ABB RAPID module: P704.mod

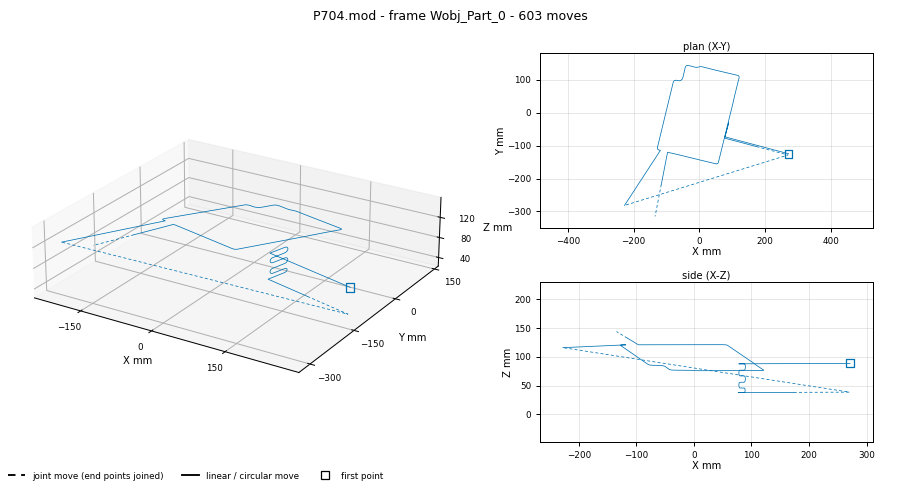
[picture p0: tool path of P704.mod in frame Wobj_Part_0, 603 of 613 moves have a stored position in this frame; points joined in program order, loops and branches not executed]
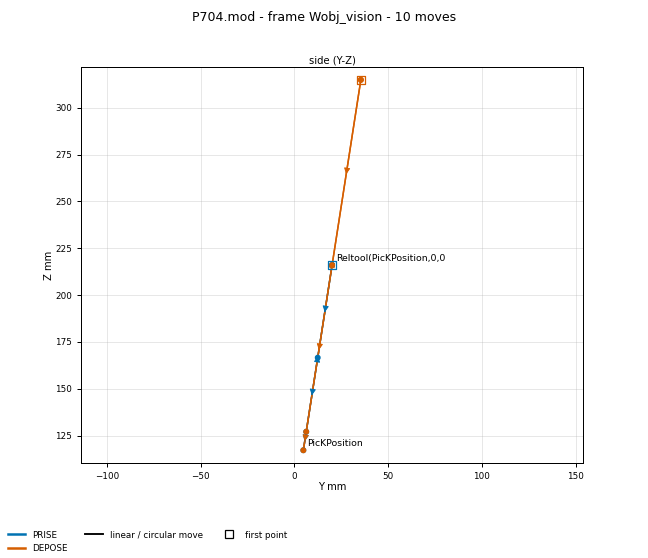
[picture p1: tool path of P704.mod in frame Wobj_vision, 10 of 613 moves have a stored position in this frame; points joined in program order, loops and branches not executed]
MODULE P704

    ! Nom         :P704
    ! Description :
    ! Créé le     :30/05/2023 09:06:17

    LOCAL CONST SPEEDDATA VitesseLente :=[10,500,0,0];
	LOCAL CONST SPEEDDATA VitesseRapide :=[30,500,0,0];
	LOCAL CONST SPEEDDATA VitesseTronconnage :=[2,500,0,0];
	LOCAL CONST SPEEDDATA VitesseTronconnageApp :=[10,500,0,0];
    !
    !Point de prise
    LOCAL PERS Robtarget PicKPosition := [[-11.2554102096367,4.78901339378507,117.207238896583],[0.0630021780734219,0.793906121478423,0.603147355662045,-0.0442387069767479],[0,0,0,0],[8.999999E+09,8.999999E+09,8.999999E+09,8.999999E+09,8.999999E+09,8.999999E+09]];
	LOCAL PERS Pose Ref := [[0,0,0],[1,0,0,0]];
    !
    !Declaration des points de meulage

    !Tr_meulage_motif_1 : Meulage d'un motif
    LOCAL CONST Robtarget Tr_meulage_motif_1_0 := [[77.98109375,-73.0847578125,87.956984375],[0.559429550316464,-0.561673578795992,-0.431884716383229,0.430159227344712],[0,0,0,0],[8.999999E+09,8.999999E+09,8.999999E+09,8.999999E+09,8.999999E+09,8.999999E+09]];
    LOCAL CONST Robtarget Tr_meulage_motif_1_1 := [[78.235953125,-72.1177734375,87.956984375],[0.559429550316464,-0.561673578795992,-0.431884716383229,0.430159227344712],[0,0,0,0],[8.999999E+09,8.999999E+09,8.999999E+09,8.999999E+09,8.999999E+09,8.999999E+09]];
    LOCAL CONST Robtarget Tr_meulage_motif_1_2 := [[78.4908046875,-71.150796875,87.956984375],[0.559429550316464,-0.561673578795992,-0.431884716383229,0.430159227344712],[0,0,0,0],[8.999999E+09,8.999999E+09,8.999999E+09,8.999999E+09,8.999999E+09,8.999999E+09]];
    LOCAL CONST Robtarget Tr_meulage_motif_1_3 := [[78.74565625,-70.1838203125,87.956984375],[0.559429550316464,-0.561673578795992,-0.431884716383229,0.430159227344712],[0,0,0,0],[8.999999E+09,8.999999E+09,8.999999E+09,8.999999E+09,8.999999E+09,8.999999E+09]];
    LOCAL CONST Robtarget Tr_meulage_motif_1_4 := [[79.0005078125,-69.2168359375,87.9569921875],[0.559429550316464,-0.561673578795992,-0.431884716383229,0.430159227344712],[0,0,0,0],[8.999999E+09,8.999999E+09,8.999999E+09,8.999999E+09,8.999999E+09,8.999999E+09]];
    LOCAL CONST Robtarget Tr_meulage_motif_1_5 := [[79.255359375,-68.249859375,87.9569921875],[0.559429550316464,-0.561673578795992,-0.431884716383229,0.430159227344712],[0,0,0,0],[8.999999E+09,8.999999E+09,8.999999E+09,8.999999E+09,8.999999E+09,8.999999E+09]];
    LOCAL CONST Robtarget Tr_meulage_motif_1_6 := [[79.51021875,-67.282875,87.9569921875],[0.559429550316464,-0.561673578795992,-0.431884716383229,0.430159227344712],[0,0,0,0],[8.999999E+09,8.999999E+09,8.999999E+09,8.999999E+09,8.999999E+09,8.999999E+09]];
    LOCAL CONST Robtarget Tr_meulage_motif_1_7 := [[79.7650703125,-66.3158984375,87.9569921875],[0.559429550316464,-0.561673578795992,-0.431884716383229,0.430159227344712],[0,0,0,0],[8.999999E+09,8.999999E+09,8.999999E+09,8.999999E+09,8.999999E+09,8.999999E+09]];
    LOCAL CONST Robtarget Tr_meulage_motif_1_8 := [[80.019921875,-65.34891796875,87.957],[0.559429550316464,-0.561673578795992,-0.431884716383229,0.430159227344712],[0,0,0,0],[8.999999E+09,8.999999E+09,8.999999E+09,8.999999E+09,8.999999E+09,8.999999E+09]];
    LOCAL CONST Robtarget Tr_meulage_motif_1_9 := [[80.2747734375,-64.38194140625,87.957],[0.559429550316464,-0.561673578795992,-0.431884716383229,0.430159227344712],[0,0,0,0],[8.999999E+09,8.999999E+09,8.999999E+09,8.999999E+09,8.999999E+09,8.999999E+09]];
    LOCAL CONST Robtarget Tr_meulage_motif_1_10 := [[80.5296328125,-63.4149609375,87.957],[0.559429550316464,-0.561673578795992,-0.431884716383229,0.430159227344712],[0,0,0,0],[8.999999E+09,8.999999E+09,8.999999E+09,8.999999E+09,8.999999E+09,8.999999E+09]];
    LOCAL CONST Robtarget Tr_meulage_motif_1_11 := [[80.784484375,-62.44798046875,87.957],[0.559429550316464,-0.561673578795992,-0.431884716383229,0.430159227344712],[0,0,0,0],[8.999999E+09,8.999999E+09,8.999999E+09,8.999999E+09,8.999999E+09,8.999999E+09]];
    LOCAL CONST Robtarget Tr_meulage_motif_1_12 := [[81.0393359375,-61.481,87.9570078125],[0.559429550316464,-0.561673578795992,-0.431884716383229,0.430159227344712],[0,0,0,0],[8.999999E+09,8.999999E+09,8.999999E+09,8.999999E+09,8.999999E+09,8.999999E+09]];
    LOCAL CONST Robtarget Tr_meulage_motif_1_13 := [[81.2941875,-60.51401953125,87.9570078125],[0.559429550316464,-0.561673578795992,-0.431884716383229,0.430159227344712],[0,0,0,0],[8.999999E+09,8.999999E+09,8.999999E+09,8.999999E+09,8.999999E+09,8.999999E+09]];
    LOCAL CONST Robtarget Tr_meulage_motif_1_14 := [[81.549046875,-59.54704296875,87.9570078125],[0.559429550316464,-0.561673578795992,-0.431884716383229,0.430159227344712],[0,0,0,0],[8.999999E+09,8.999999E+09,8.999999E+09,8.999999E+09,8.999999E+09,8.999999E+09]];
    LOCAL CONST Robtarget Tr_meulage_motif_1_15 := [[81.8038984375,-58.5800625,87.9570078125],[0.559429550316464,-0.561673578795992,-0.431884716383229,0.430159227344712],[0,0,0,0],[8.999999E+09,8.999999E+09,8.999999E+09,8.999999E+09,8.999999E+09,8.999999E+09]];
    LOCAL CONST Robtarget Tr_meulage_motif_1_16 := [[82.05875,-57.61308203125,87.957015625],[0.559429550316464,-0.561673578795992,-0.431884716383229,0.430159227344712],[0,0,0,0],[8.999999E+09,8.999999E+09,8.999999E+09,8.999999E+09,8.999999E+09,8.999999E+09]];
    LOCAL CONST Robtarget Tr_meulage_motif_1_17 := [[82.3136015625,-56.6461015625,87.957015625],[0.559429550316464,-0.561673578795992,-0.431884716383229,0.430159227344712],[0,0,0,0],[8.999999E+09,8.999999E+09,8.999999E+09,8.999999E+09,8.999999E+09,8.999999E+09]];
    LOCAL CONST Robtarget Tr_meulage_motif_1_18 := [[82.5684609375,-55.67912109375,87.957015625],[0.559429550316464,-0.561673578795992,-0.431884716383229,0.430159227344712],[0,0,0,0],[8.999999E+09,8.999999E+09,8.999999E+09,8.999999E+09,8.999999E+09,8.999999E+09]];
    LOCAL CONST Robtarget Tr_meulage_motif_1_19 := [[82.8233125,-54.712140625,87.957015625],[0.559429550316464,-0.561673578795992,-0.431884716383229,0.430159227344712],[0,0,0,0],[8.999999E+09,8.999999E+09,8.999999E+09,8.999999E+09,8.999999E+09,8.999999E+09]];
    LOCAL CONST Robtarget Tr_meulage_motif_1_20 := [[83.0781640625,-53.7451640625,87.9570234375],[0.559429550316464,-0.561673578795992,-0.431884716383229,0.430159227344712],[0,0,0,0],[8.999999E+09,8.999999E+09,8.999999E+09,8.999999E+09,8.999999E+09,8.999999E+09]];
    LOCAL CONST Robtarget Tr_meulage_motif_1_21 := [[83.333015625,-52.77818359375,87.9570234375],[0.559429550316464,-0.561673578795992,-0.431884716383229,0.430159227344712],[0,0,0,0],[8.999999E+09,8.999999E+09,8.999999E+09,8.999999E+09,8.999999E+09,8.999999E+09]];
    LOCAL CONST Robtarget Tr_meulage_motif_1_22 := [[83.587875,-51.811203125,87.9570234375],[0.559429550316464,-0.561673578795992,-0.431884716383229,0.430159227344712],[0,0,0,0],[8.999999E+09,8.999999E+09,8.999999E+09,8.999999E+09,8.999999E+09,8.999999E+09]];
    LOCAL CONST Robtarget Tr_meulage_motif_1_23 := [[83.8427265625,-50.84422265625,87.9570234375],[0.559429550316464,-0.561673578795992,-0.431884716383229,0.430159227344712],[0,0,0,0],[8.999999E+09,8.999999E+09,8.999999E+09,8.999999E+09,8.999999E+09,8.999999E+09]];
    LOCAL CONST Robtarget Tr_meulage_motif_1_24 := [[84.097578125,-49.8772421875,87.95703125],[0.559429550316464,-0.561673578795992,-0.431884716383229,0.430159227344712],[0,0,0,0],[8.999999E+09,8.999999E+09,8.999999E+09,8.999999E+09,8.999999E+09,8.999999E+09]];
    LOCAL CONST Robtarget Tr_meulage_motif_1_25 := [[84.3524296875,-48.910265625,87.95703125],[0.559429550316464,-0.561673578795992,-0.431884716383229,0.430159227344712],[0,0,0,0],[8.999999E+09,8.999999E+09,8.999999E+09,8.999999E+09,8.999999E+09,8.999999E+09]];
    LOCAL CONST Robtarget Tr_meulage_motif_1_26 := [[84.60728125,-47.94328515625,87.95703125],[0.559429550316464,-0.561673578795992,-0.431884716383229,0.430159227344712],[0,0,0,0],[8.999999E+09,8.999999E+09,8.999999E+09,8.999999E+09,8.999999E+09,8.999999E+09]];
    LOCAL CONST Robtarget Tr_meulage_motif_1_27 := [[84.862140625,-46.9763046875,87.95703125],[0.559429550316464,-0.561673578795992,-0.431884716383229,0.430159227344712],[0,0,0,0],[8.999999E+09,8.999999E+09,8.999999E+09,8.999999E+09,8.999999E+09,8.999999E+09]];
    LOCAL CONST Robtarget Tr_meulage_motif_1_28 := [[85.1169921875,-46.00932421875,87.9570390625],[0.559429550316464,-0.561673578795992,-0.431884716383229,0.430159227344712],[0,0,0,0],[8.999999E+09,8.999999E+09,8.999999E+09,8.999999E+09,8.999999E+09,8.999999E+09]];
    LOCAL CONST Robtarget Tr_meulage_motif_1_29 := [[85.37184375,-45.04234375,87.9570390625],[0.559429550316464,-0.561673578795992,-0.431884716383229,0.430159227344712],[0,0,0,0],[8.999999E+09,8.999999E+09,8.999999E+09,8.999999E+09,8.999999E+09,8.999999E+09]];
    LOCAL CONST Robtarget Tr_meulage_motif_1_30 := [[85.6266953125,-44.0753671875,87.9570390625],[0.559429550316464,-0.561673578795992,-0.431884716383229,0.430159227344712],[0,0,0,0],[8.999999E+09,8.999999E+09,8.999999E+09,8.999999E+09,8.999999E+09,8.999999E+09]];
    LOCAL CONST Robtarget Tr_meulage_motif_1_31 := [[85.8815546875,-43.10838671875,87.9570390625],[0.559429550316464,-0.561673578795992,-0.431884716383229,0.430159227344712],[0,0,0,0],[8.999999E+09,8.999999E+09,8.999999E+09,8.999999E+09,8.999999E+09,8.999999E+09]];
    LOCAL CONST Robtarget Tr_meulage_motif_1_32 := [[86.13640625,-42.14140625,87.957046875],[0.559429550316464,-0.561673578795992,-0.431884716383229,0.430159227344712],[0,0,0,0],[8.999999E+09,8.999999E+09,8.999999E+09,8.999999E+09,8.999999E+09,8.999999E+09]];
    LOCAL CONST Robtarget Tr_meulage_motif_1_33 := [[86.3912578125,-41.17442578125,87.957046875],[0.559429550316464,-0.561673578795992,-0.431884716383229,0.430159227344712],[0,0,0,0],[8.999999E+09,8.999999E+09,8.999999E+09,8.999999E+09,8.999999E+09,8.999999E+09]];
    LOCAL CONST Robtarget Tr_meulage_motif_1_34 := [[86.646109375,-40.2074453125,87.957046875],[0.559429550316464,-0.561673578795992,-0.431884716383229,0.430159227344712],[0,0,0,0],[8.999999E+09,8.999999E+09,8.999999E+09,8.999999E+09,8.999999E+09,8.999999E+09]];
    LOCAL CONST Robtarget Tr_meulage_motif_1_35 := [[86.90096875,-39.24046875,87.957046875],[0.559429550316464,-0.561673578795992,-0.431884716383229,0.430159227344712],[0,0,0,0],[8.999999E+09,8.999999E+09,8.999999E+09,8.999999E+09,8.999999E+09,8.999999E+09]];
    LOCAL CONST Robtarget Tr_meulage_motif_1_36 := [[87.1558203125,-38.27348828125,87.9570546875],[0.559429550316464,-0.561673578795992,-0.431884716383229,0.430159227344712],[0,0,0,0],[8.999999E+09,8.999999E+09,8.999999E+09,8.999999E+09,8.999999E+09,8.999999E+09]];
    LOCAL CONST Robtarget Tr_meulage_motif_1_37 := [[87.410671875,-37.3065078125,87.9570546875],[0.559429550316464,-0.561673578795992,-0.431884716383229,0.430159227344712],[0,0,0,0],[8.999999E+09,8.999999E+09,8.999999E+09,8.999999E+09,8.999999E+09,8.999999E+09]];
    LOCAL CONST Robtarget Tr_meulage_motif_1_38 := [[87.6655234375,-36.33952734375,87.9570546875],[0.559429550316464,-0.561673578795992,-0.431884716383229,0.430159227344712],[0,0,0,0],[8.999999E+09,8.999999E+09,8.999999E+09,8.999999E+09,8.999999E+09,8.999999E+09]];
    LOCAL CONST Robtarget Tr_meulage_motif_1_39 := [[87.9182109375,-35.37966796875,87.8464609375],[0.559429550316464,-0.561673578795992,-0.431884716383229,0.430159227344712],[0,0,0,0],[8.999999E+09,8.999999E+09,8.999999E+09,8.999999E+09,8.999999E+09,8.999999E+09]];
    LOCAL CONST Robtarget Tr_meulage_motif_1_40 := [[88.158921875,-34.4642890625,87.63528125],[0.559429550316464,-0.561673578795992,-0.431884716383229,0.430159227344712],[0,0,0,0],[8.999999E+09,8.999999E+09,8.999999E+09,8.999999E+09,8.999999E+09,8.999999E+09]];
    LOCAL CONST Robtarget Tr_meulage_motif_1_41 := [[88.375578125,-33.63955078125,87.3634375],[0.559429550316464,-0.561673578795992,-0.431884716383229,0.430159227344712],[0,0,0,0],[8.999999E+09,8.999999E+09,8.999999E+09,8.999999E+09,8.999999E+09,8.999999E+09]];
    LOCAL CONST Robtarget Tr_meulage_motif_1_42 := [[88.56603125,-32.91419921875,87.0875],[0.559429550316464,-0.561673578795992,-0.431884716383229,0.430159227344712],[0,0,0,0],[8.999999E+09,8.999999E+09,8.999999E+09,8.999999E+09,8.999999E+09,8.999999E+09]];
    LOCAL CONST Robtarget Tr_meulage_motif_1_43 := [[88.845140625,-31.84909765625,86.4713828125],[0.559429550316464,-0.561673578795992,-0.431884716383229,0.430159227344712],[0,0,0,0],[8.999999E+09,8.999999E+09,8.999999E+09,8.999999E+09,8.999999E+09,8.999999E+09]];
    LOCAL CONST Robtarget Tr_meulage_motif_1_44 := [[89.104015625,-30.858484375,85.623734375],[0.559429550316464,-0.561673578795992,-0.431884716383229,0.430159227344712],[0,0,0,0],[8.999999E+09,8.999999E+09,8.999999E+09,8.999999E+09,8.999999E+09,8.999999E+09]];
    LOCAL CONST Robtarget Tr_meulage_motif_1_45 := [[89.317546875,-30.03816015625,84.599859375],[0.559429550316464,-0.561673578795992,-0.431884716383229,0.430159227344712],[0,0,0,0],[8.999999E+09,8.999999E+09,8.999999E+09,8.999999E+09,8.999999E+09,8.999999E+09]];
    LOCAL CONST Robtarget Tr_meulage_motif_1_46 := [[89.4392421875,-29.565404296875,83.4836796875],[0.559429550316464,-0.561673578795992,-0.431884716383229,0.430159227344712],[0,0,0,0],[8.999999E+09,8.999999E+09,8.999999E+09,8.999999E+09,8.999999E+09,8.999999E+09]];
    LOCAL CONST Robtarget Tr_meulage_motif_1_47 := [[89.4444453125,-29.538787109375,82.7877109375],[0.559429550316464,-0.561673578795992,-0.431884716383229,0.430159227344712],[0,0,0,0],[8.999999E+09,8.999999E+09,8.999999E+09,8.999999E+09,8.999999E+09,8.999999E+09]];
    LOCAL CONST Robtarget Tr_meulage_motif_1_48 := [[89.4428359375,-29.538361328125,82.1264609375],[0.559429550316464,-0.561673578795992,-0.431884716383229,0.430159227344712],[0,0,0,0],[8.999999E+09,8.999999E+09,8.999999E+09,8.999999E+09,8.999999E+09,8.999999E+09]];
    LOCAL CONST Robtarget Tr_meulage_motif_1_49 := [[89.427234375,-29.591,81.465375],[0.559429550316464,-0.561673578795992,-0.431884716383229,0.430159227344712],[0,0,0,0],[8.999999E+09,8.999999E+09,8.999999E+09,8.999999E+09,8.999999E+09,8.999999E+09]];
    LOCAL CONST Robtarget Tr_meulage_motif_1_50 := [[89.2975859375,-30.07205859375,80.363625],[0.559429550316464,-0.561673578795992,-0.431884716383229,0.430159227344712],[0,0,0,0],[8.999999E+09,8.999999E+09,8.999999E+09,8.999999E+09,8.999999E+09,8.999999E+09]];
    LOCAL CONST Robtarget Tr_meulage_motif_1_51 := [[89.0768203125,-30.899748046875,79.357],[0.559429550316464,-0.561673578795992,-0.431884716383229,0.430159227344712],[0,0,0,0],[8.999999E+09,8.999999E+09,8.999999E+09,8.999999E+09,8.999999E+09,8.999999E+09]];
    LOCAL CONST Robtarget Tr_meulage_motif_1_52 := [[88.813984375,-31.888828125,78.528125],[0.559429550316464,-0.561673578795992,-0.431884716383229,0.430159227344712],[0,0,0,0],[8.999999E+09,8.999999E+09,8.999999E+09,8.999999E+09,8.999999E+09,8.999999E+09]];
    LOCAL CONST Robtarget Tr_meulage_motif_1_53 := [[88.6379140625,-32.552978515625,78.132375],[0.559429550316464,-0.561673578795992,-0.431884716383229,0.430159227344712],[0,0,0,0],[8.999999E+09,8.999999E+09,8.999999E+09,8.999999E+09,8.999999E+09,8.999999E+09]];
    LOCAL CONST Robtarget Tr_meulage_motif_1_54 := [[88.3415625,-33.672578125,77.64484375],[0.559429550316464,-0.561673578795992,-0.431884716383229,0.430159227344712],[0,0,0,0],[8.999999E+09,8.999999E+09,8.999999E+09,8.999999E+09,8.999999E+09,8.999999E+09]];
    LOCAL CONST Robtarget Tr_meulage_motif_1_55 := [[88.1255625,-34.4895390625,77.38075],[0.559429550316464,-0.561673578795992,-0.431884716383229,0.430159227344712],[0,0,0,0],[8.999999E+09,8.999999E+09,8.999999E+09,8.999999E+09,8.999999E+09,8.999999E+09]];
    LOCAL CONST Robtarget Tr_meulage_motif_1_56 := [[87.8875390625,-35.39062890625,77.17628125],[0.559429550316464,-0.561673578795992,-0.431884716383229,0.430159227344712],[0,0,0,0],[8.999999E+09,8.999999E+09,8.999999E+09,8.999999E+09,8.999999E+09,8.999999E+09]];
    LOCAL CONST Robtarget Tr_meulage_motif_1_57 := [[87.637125,-36.3397109375,77.0676875],[0.559429550316464,-0.561673578795992,-0.431884716383229,0.430159227344712],[0,0,0,0],[8.999999E+09,8.999999E+09,8.999999E+09,8.999999E+09,8.999999E+09,8.999999E+09]];
    LOCAL CONST Robtarget Tr_meulage_motif_1_58 := [[87.3838984375,-37.2994296875,76.9570859375],[0.559429550316464,-0.561673578795992,-0.431884716383229,0.430159227344712],[0,0,0,0],[8.999999E+09,8.999999E+09,8.999999E+09,8.999999E+09,8.999999E+09,8.999999E+09]];
    LOCAL CONST Robtarget Tr_meulage_motif_1_59 := [[87.1290390625,-38.26641015625,76.9570859375],[0.559429550316464,-0.561673578795992,-0.431884716383229,0.430159227344712],[0,0,0,0],[8.999999E+09,8.999999E+09,8.999999E+09,8.999999E+09,8.999999E+09,8.999999E+09]];
    LOCAL CONST Robtarget Tr_meulage_motif_1_60 := [[86.8741875,-39.23338671875,76.9570859375],[0.559429550316464,-0.561673578795992,-0.431884716383229,0.430159227344712],[0,0,0,0],[8.999999E+09,8.999999E+09,8.999999E+09,8.999999E+09,8.999999E+09,8.999999E+09]];
    LOCAL CONST Robtarget Tr_meulage_motif_1_61 := [[86.6193359375,-40.2003671875,76.9570859375],[0.559429550316464,-0.561673578795992,-0.431884716383229,0.430159227344712],[0,0,0,0],[8.999999E+09,8.999999E+09,8.999999E+09,8.999999E+09,8.999999E+09,8.999999E+09]];
    LOCAL CONST Robtarget Tr_meulage_motif_1_62 := [[86.364484375,-41.16734765625,76.957078125],[0.559429550316464,-0.561673578795992,-0.431884716383229,0.430159227344712],[0,0,0,0],[8.999999E+09,8.999999E+09,8.999999E+09,8.999999E+09,8.999999E+09,8.999999E+09]];
    LOCAL CONST Robtarget Tr_meulage_motif_1_63 := [[86.109625,-42.134328125,76.957078125],[0.559429550316464,-0.561673578795992,-0.431884716383229,0.430159227344712],[0,0,0,0],[8.999999E+09,8.999999E+09,8.999999E+09,8.999999E+09,8.999999E+09,8.999999E+09]];
    LOCAL CONST Robtarget Tr_meulage_motif_1_64 := [[85.8547734375,-43.10130859375,76.957078125],[0.559429550316464,-0.561673578795992,-0.431884716383229,0.430159227344712],[0,0,0,0],[8.999999E+09,8.999999E+09,8.999999E+09,8.999999E+09,8.999999E+09,8.999999E+09]];
    LOCAL CONST Robtarget Tr_meulage_motif_1_65 := [[85.599921875,-44.06828515625,76.957078125],[0.559429550316464,-0.561673578795992,-0.431884716383229,0.430159227344712],[0,0,0,0],[8.999999E+09,8.999999E+09,8.999999E+09,8.999999E+09,8.999999E+09,8.999999E+09]];
    LOCAL CONST Robtarget Tr_meulage_motif_1_66 := [[85.3450703125,-45.035265625,76.9570703125],[0.559429550316464,-0.561673578795992,-0.431884716383229,0.430159227344712],[0,0,0,0],[8.999999E+09,8.999999E+09,8.999999E+09,8.999999E+09,8.999999E+09,8.999999E+09]];
    LOCAL CONST Robtarget Tr_meulage_motif_1_67 := [[85.0902109375,-46.00224609375,76.9570703125],[0.559429550316464,-0.561673578795992,-0.431884716383229,0.430159227344712],[0,0,0,0],[8.999999E+09,8.999999E+09,8.999999E+09,8.999999E+09,8.999999E+09,8.999999E+09]];
    LOCAL CONST Robtarget Tr_meulage_motif_1_68 := [[84.835359375,-46.9692265625,76.9570703125],[0.559429550316464,-0.561673578795992,-0.431884716383229,0.430159227344712],[0,0,0,0],[8.999999E+09,8.999999E+09,8.999999E+09,8.999999E+09,8.999999E+09,8.999999E+09]];
    LOCAL CONST Robtarget Tr_meulage_motif_1_69 := [[84.5805078125,-47.93620703125,76.9570703125],[0.559429550316464,-0.561673578795992,-0.431884716383229,0.430159227344712],[0,0,0,0],[8.999999E+09,8.999999E+09,8.999999E+09,8.999999E+09,8.999999E+09,8.999999E+09]];
    LOCAL CONST Robtarget Tr_meulage_motif_1_70 := [[84.32565625,-48.90318359375,76.9570625],[0.559429550316464,-0.561673578795992,-0.431884716383229,0.430159227344712],[0,0,0,0],[8.999999E+09,8.999999E+09,8.999999E+09,8.999999E+09,8.999999E+09,8.999999E+09]];
    LOCAL CONST Robtarget Tr_meulage_motif_1_71 := [[84.070796875,-49.8701640625,76.9570625],[0.559429550316464,-0.561673578795992,-0.431884716383229,0.430159227344712],[0,0,0,0],[8.999999E+09,8.999999E+09,8.999999E+09,8.999999E+09,8.999999E+09,8.999999E+09]];
    LOCAL CONST Robtarget Tr_meulage_motif_1_72 := [[83.8159453125,-50.83714453125,76.9570625],[0.559429550316464,-0.561673578795992,-0.431884716383229,0.430159227344712],[0,0,0,0],[8.999999E+09,8.999999E+09,8.999999E+09,8.999999E+09,8.999999E+09,8.999999E+09]];
    LOCAL CONST Robtarget Tr_meulage_motif_1_73 := [[83.56109375,-51.804125,76.9570625],[0.559429550316464,-0.561673578795992,-0.431884716383229,0.430159227344712],[0,0,0,0],[8.999999E+09,8.999999E+09,8.999999E+09,8.999999E+09,8.999999E+09,8.999999E+09]];
    LOCAL CONST Robtarget Tr_meulage_motif_1_74 := [[83.3062421875,-52.77110546875,76.9570546875],[0.559429550316464,-0.561673578795992,-0.431884716383229,0.430159227344712],[0,0,0,0],[8.999999E+09,8.999999E+09,8.999999E+09,8.999999E+09,8.999999E+09,8.999999E+09]];
    LOCAL CONST Robtarget Tr_meulage_motif_1_75 := [[83.051390625,-53.73808203125,76.9570546875],[0.559429550316464,-0.561673578795992,-0.431884716383229,0.430159227344712],[0,0,0,0],[8.999999E+09,8.999999E+09,8.999999E+09,8.999999E+09,8.999999E+09,8.999999E+09]];
    LOCAL CONST Robtarget Tr_meulage_motif_1_76 := [[82.79653125,-54.7050625,76.9570546875],[0.559429550316464,-0.561673578795992,-0.431884716383229,0.430159227344712],[0,0,0,0],[8.999999E+09,8.999999E+09,8.999999E+09,8.999999E+09,8.999999E+09,8.999999E+09]];
    LOCAL CONST Robtarget Tr_meulage_motif_1_77 := [[82.5416796875,-55.67204296875,76.9570546875],[0.559429550316464,-0.561673578795992,-0.431884716383229,0.430159227344712],[0,0,0,0],[8.999999E+09,8.999999E+09,8.999999E+09,8.999999E+09,8.999999E+09,8.999999E+09]];
    LOCAL CONST Robtarget Tr_meulage_motif_1_78 := [[82.286828125,-56.6390234375,76.957046875],[0.559429550316464,-0.561673578795992,-0.431884716383229,0.430159227344712],[0,0,0,0],[8.999999E+09,8.999999E+09,8.999999E+09,8.999999E+09,8.999999E+09,8.999999E+09]];
    LOCAL CONST Robtarget Tr_meulage_motif_1_79 := [[82.0319765625,-57.60600390625,76.957046875],[0.559429550316464,-0.561673578795992,-0.431884716383229,0.430159227344712],[0,0,0,0],[8.999999E+09,8.999999E+09,8.999999E+09,8.999999E+09,8.999999E+09,8.999999E+09]];
    LOCAL CONST Robtarget Tr_meulage_motif_1_80 := [[81.7771171875,-58.57298046875,76.957046875],[0.559429550316464,-0.561673578795992,-0.431884716383229,0.430159227344712],[0,0,0,0],[8.999999E+09,8.999999E+09,8.999999E+09,8.999999E+09,8.999999E+09,8.999999E+09]];
    LOCAL CONST Robtarget Tr_meulage_motif_1_81 := [[81.522265625,-59.5399609375,76.957046875],[0.559429550316464,-0.561673578795992,-0.431884716383229,0.430159227344712],[0,0,0,0],[8.999999E+09,8.999999E+09,8.999999E+09,8.999999E+09,8.999999E+09,8.999999E+09]];
    LOCAL CONST Robtarget Tr_meulage_motif_1_82 := [[81.2674140625,-60.50694140625,76.9570390625],[0.559429550316464,-0.561673578795992,-0.431884716383229,0.430159227344712],[0,0,0,0],[8.999999E+09,8.999999E+09,8.999999E+09,8.999999E+09,8.999999E+09,8.999999E+09]];
    LOCAL CONST Robtarget Tr_meulage_motif_1_83 := [[81.0125625,-61.473921875,76.9570390625],[0.559429550316464,-0.561673578795992,-0.431884716383229,0.430159227344712],[0,0,0,0],[8.999999E+09,8.999999E+09,8.999999E+09,8.999999E+09,8.999999E+09,8.999999E+09]];
    LOCAL CONST Robtarget Tr_meulage_motif_1_84 := [[80.757703125,-62.44090234375,76.9570390625],[0.559429550316464,-0.561673578795992,-0.431884716383229,0.430159227344712],[0,0,0,0],[8.999999E+09,8.999999E+09,8.999999E+09,8.999999E+09,8.999999E+09,8.999999E+09]];
    LOCAL CONST Robtarget Tr_meulage_motif_1_85 := [[80.5028515625,-63.40787890625,76.9570390625],[0.559429550316464,-0.561673578795992,-0.431884716383229,0.430159227344712],[0,0,0,0],[8.999999E+09,8.999999E+09,8.999999E+09,8.999999E+09,8.999999E+09,8.999999E+09]];
    LOCAL CONST Robtarget Tr_meulage_motif_1_86 := [[80.248,-64.374859375,76.95703125],[0.559429550316464,-0.561673578795992,-0.431884716383229,0.430159227344712],[0,0,0,0],[8.999999E+09,8.999999E+09,8.999999E+09,8.999999E+09,8.999999E+09,8.999999E+09]];
    LOCAL CONST Robtarget Tr_meulage_motif_1_87 := [[79.9931484375,-65.34183984375,76.95703125],[0.559429550316464,-0.561673578795992,-0.431884716383229,0.430159227344712],[0,0,0,0],[8.999999E+09,8.999999E+09,8.999999E+09,8.999999E+09,8.999999E+09,8.999999E+09]];
    LOCAL CONST Robtarget Tr_meulage_motif_1_88 := [[79.7382890625,-66.3088203125,76.95703125],[0.559429550316464,-0.561673578795992,-0.431884716383229,0.430159227344712],[0,0,0,0],[8.999999E+09,8.999999E+09,8.999999E+09,8.999999E+09,8.999999E+09,8.999999E+09]];
    LOCAL CONST Robtarget Tr_meulage_motif_1_89 := [[79.4850625,-67.2685390625,76.8464375],[0.559429550316464,-0.561673578795992,-0.431884716383229,0.430159227344712],[0,0,0,0],[8.999999E+09,8.999999E+09,8.999999E+09,8.999999E+09,8.999999E+09,8.999999E+09]];
    LOCAL CONST Robtarget Tr_meulage_motif_1_90 := [[79.2433359375,-68.1836484375,76.63525],[0.559429550316464,-0.561673578795992,-0.431884716383229,0.430159227344712],[0,0,0,0],[8.999999E+09,8.999999E+09,8.999999E+09,8.999999E+09,8.999999E+09,8.999999E+09]];
    LOCAL CONST Robtarget Tr_meulage_motif_1_91 := [[79.0253515625,-69.00803125,76.36340625],[0.559429550316464,-0.561673578795992,-0.431884716383229,0.430159227344712],[0,0,0,0],[8.999999E+09,8.999999E+09,8.999999E+09,8.999999E+09,8.999999E+09,8.999999E+09]];
    LOCAL CONST Robtarget Tr_meulage_motif_1_92 := [[78.84328125,-69.69584375,76.0592421875],[0.559429550316464,-0.561673578795992,-0.431884716383229,0.430159227344712],[0,0,0,0],[8.999999E+09,8.999999E+09,8.999999E+09,8.999999E+09,8.999999E+09,8.999999E+09]];
    LOCAL CONST Robtarget Tr_meulage_motif_1_93 := [[78.57803125,-70.6957265625,75.3967109375],[0.559429550316464,-0.561673578795992,-0.431884716383229,0.430159227344712],[0,0,0,0],[8.999999E+09,8.999999E+09,8.999999E+09,8.999999E+09,8.999999E+09,8.999999E+09]];
    LOCAL CONST Robtarget Tr_meulage_motif_1_94 := [[78.3459765625,-71.5673046875,74.49478125],[0.559429550316464,-0.561673578795992,-0.431884716383229,0.430159227344712],[0,0,0,0],[8.999999E+09,8.999999E+09,8.999999E+09,8.999999E+09,8.999999E+09,8.999999E+09]];
    LOCAL CONST Robtarget Tr_meulage_motif_1_95 := [[78.20709375,-72.0839296875,73.44875],[0.559429550316464,-0.561673578795992,-0.431884716383229,0.430159227344712],[0,0,0,0],[8.999999E+09,8.999999E+09,8.999999E+09,8.999999E+09,8.999999E+09,8.999999E+09]];
    LOCAL CONST Robtarget Tr_meulage_motif_1_96 := [[78.1583125,-72.2621640625,72.75553125],[0.559429550316464,-0.561673578795992,-0.431884716383229,0.430159227344712],[0,0,0,0],[8.999999E+09,8.999999E+09,8.999999E+09,8.999999E+09,8.999999E+09,8.999999E+09]];
    LOCAL CONST Robtarget Tr_meulage_motif_1_97 := [[78.1401640625,-72.32340625,71.98553125],[0.559429550316464,-0.561673578795992,-0.431884716383229,0.430159227344712],[0,0,0,0],[8.999999E+09,8.999999E+09,8.999999E+09,8.999999E+09,8.999999E+09,8.999999E+09]];
    LOCAL CONST Robtarget Tr_meulage_motif_1_98 := [[78.1553515625,-72.2581875,71.2156640625],[0.559429550316464,-0.561673578795992,-0.431884716383229,0.430159227344712],[0,0,0,0],[8.999999E+09,8.999999E+09,8.999999E+09,8.999999E+09,8.999999E+09,8.999999E+09]];
    LOCAL CONST Robtarget Tr_meulage_motif_1_99 := [[78.2595859375,-71.851734375,70.1074140625],[0.559429550316464,-0.561673578795992,-0.431884716383229,0.430159227344712],[0,0,0,0],[8.999999E+09,8.999999E+09,8.999999E+09,8.999999E+09,8.999999E+09,8.999999E+09]];
    LOCAL CONST Robtarget Tr_meulage_motif_1_100 := [[78.36375,-71.4507265625,69.521734375],[0.559429550316464,-0.561673578795992,-0.431884716383229,0.430159227344712],[0,0,0,0],[8.999999E+09,8.999999E+09,8.999999E+09,8.999999E+09,8.999999E+09,8.999999E+09]];
    LOCAL CONST Robtarget Tr_meulage_motif_1_101 := [[78.5876796875,-70.5923203125,68.634609375],[0.559429550316464,-0.561673578795992,-0.431884716383229,0.430159227344712],[0,0,0,0],[8.999999E+09,8.999999E+09,8.999999E+09,8.999999E+09,8.999999E+09,8.999999E+09]];
    LOCAL CONST Robtarget Tr_meulage_motif_1_102 := [[78.7359375,-70.025703125,68.2203046875],[0.559429550316464,-0.561673578795992,-0.431884716383229,0.430159227344712],[0,0,0,0],[8.999999E+09,8.999999E+09,8.999999E+09,8.999999E+09,8.999999E+09,8.999999E+09]];
    LOCAL CONST Robtarget Tr_meulage_motif_1_103 := [[79.019515625,-68.944359375,67.6762109375],[0.559429550316464,-0.561673578795992,-0.431884716383229,0.430159227344712],[0,0,0,0],[8.999999E+09,8.999999E+09,8.999999E+09,8.999999E+09,8.999999E+09,8.999999E+09]];
    LOCAL CONST Robtarget Tr_meulage_motif_1_104 := [[79.2291953125,-68.14584375,67.3807109375],[0.559429550316464,-0.561673578795992,-0.431884716383229,0.430159227344712],[0,0,0,0],[8.999999E+09,8.999999E+09,8.999999E+09,8.999999E+09,8.999999E+09,8.999999E+09]];
    LOCAL CONST Robtarget Tr_meulage_motif_1_105 := [[79.4662265625,-67.244484375,67.17625],[0.559429550316464,-0.561673578795992,-0.431884716383229,0.430159227344712],[0,0,0,0],[8.999999E+09,8.999999E+09,8.999999E+09,8.999999E+09,8.999999E+09,8.999999E+09]];
    LOCAL CONST Robtarget Tr_meulage_motif_1_106 := [[79.7161171875,-66.295265625,67.06765625],[0.559429550316464,-0.561673578795992,-0.431884716383229,0.430159227344712],[0,0,0,0],[8.999999E+09,8.999999E+09,8.999999E+09,8.999999E+09,8.999999E+09,8.999999E+09]];
    LOCAL CONST Robtarget Tr_meulage_motif_1_107 := [[79.9688046875,-65.33540234375,66.9570625],[0.559429550316464,-0.561673578795992,-0.431884716383229,0.430159227344712],[0,0,0,0],[8.999999E+09,8.999999E+09,8.999999E+09,8.999999E+09,8.999999E+09,8.999999E+09]];
    LOCAL CONST Robtarget Tr_meulage_motif_1_108 := [[80.22365625,-64.36842578125,66.9570703125],[0.559429550316464,-0.561673578795992,-0.431884716383229,0.430159227344712],[0,0,0,0],[8.999999E+09,8.999999E+09,8.999999E+09,8.999999E+09,8.999999E+09,8.999999E+09]];
    LOCAL CONST Robtarget Tr_meulage_motif_1_109 := [[80.4785078125,-63.4014453125,66.9570703125],[0.559429550316464,-0.561673578795992,-0.431884716383229,0.430159227344712],[0,0,0,0],[8.999999E+09,8.999999E+09,8.999999E+09,8.999999E+09,8.999999E+09,8.999999E+09]];
    LOCAL CONST Robtarget Tr_meulage_motif_1_110 := [[80.733359375,-62.43446484375,66.9570703125],[0.559429550316464,-0.561673578795992,-0.431884716383229,0.430159227344712],[0,0,0,0],[8.999999E+09,8.999999E+09,8.999999E+09,8.999999E+09,8.999999E+09,8.999999E+09]];
    LOCAL CONST Robtarget Tr_meulage_motif_1_111 := [[80.98821875,-61.467484375,66.9570703125],[0.559429550316464,-0.561673578795992,-0.431884716383229,0.430159227344712],[0,0,0,0],[8.999999E+09,8.999999E+09,8.999999E+09,8.999999E+09,8.999999E+09,8.999999E+09]];
    LOCAL CONST Robtarget Tr_meulage_motif_1_112 := [[81.2430703125,-60.50050390625,66.957078125],[0.559429550316464,-0.561673578795992,-0.431884716383229,0.430159227344712],[0,0,0,0],[8.999999E+09,8.999999E+09,8.999999E+09,8.999999E+09,8.999999E+09,8.999999E+09]];
    LOCAL CONST Robtarget Tr_meulage_motif_1_113 := [[81.497921875,-59.53352734375,66.957078125],[0.559429550316464,-0.561673578795992,-0.431884716383229,0.430159227344712],[0,0,0,0],[8.999999E+09,8.999999E+09,8.999999E+09,8.999999E+09,8.999999E+09,8.999999E+09]];
    LOCAL CONST Robtarget Tr_meulage_motif_1_114 := [[81.7527734375,-58.566546875,66.957078125],[0.559429550316464,-0.561673578795992,-0.431884716383229,0.430159227344712],[0,0,0,0],[8.999999E+09,8.999999E+09,8.999999E+09,8.999999E+09,8.999999E+09,8.999999E+09]];
    LOCAL CONST Robtarget Tr_meulage_motif_1_115 := [[82.0076328125,-57.59956640625,66.957078125],[0.559429550316464,-0.561673578795992,-0.431884716383229,0.430159227344712],[0,0,0,0],[8.999999E+09,8.999999E+09,8.999999E+09,8.999999E+09,8.999999E+09,8.999999E+09]];
    LOCAL CONST Robtarget Tr_meulage_motif_1_116 := [[82.262484375,-56.6325859375,66.9570859375],[0.559429550316464,-0.561673578795992,-0.431884716383229,0.430159227344712],[0,0,0,0],[8.999999E+09,8.999999E+09,8.999999E+09,8.999999E+09,8.999999E+09,8.999999E+09]];
    LOCAL CONST Robtarget Tr_meulage_motif_1_117 := [[82.5173359375,-55.66560546875,66.9570859375],[0.559429550316464,-0.561673578795992,-0.431884716383229,0.430159227344712],[0,0,0,0],[8.999999E+09,8.999999E+09,8.999999E+09,8.999999E+09,8.999999E+09,8.999999E+09]];
    LOCAL CONST Robtarget Tr_meulage_motif_1_118 := [[82.7721875,-54.69862890625,66.9570859375],[0.559429550316464,-0.561673578795992,-0.431884716383229,0.430159227344712],[0,0,0,0],[8.999999E+09,8.999999E+09,8.999999E+09,8.999999E+09,8.999999E+09,8.999999E+09]];
    LOCAL CONST Robtarget Tr_meulage_motif_1_119 := [[83.027046875,-53.7316484375,66.9570859375],[0.559429550316464,-0.561673578795992,-0.431884716383229,0.430159227344712],[0,0,0,0],[8.999999E+09,8.999999E+09,8.999999E+09,8.999999E+09,8.999999E+09,8.999999E+09]];
    LOCAL CONST Robtarget Tr_meulage_motif_1_120 := [[83.2818984375,-52.76466796875,66.9570859375],[0.559429550316464,-0.561673578795992,-0.431884716383229,0.430159227344712],[0,0,0,0],[8.999999E+09,8.999999E+09,8.999999E+09,8.999999E+09,8.999999E+09,8.999999E+09]];
    LOCAL CONST Robtarget Tr_meulage_motif_1_121 := [[83.53675,-51.7976875,66.95709375],[0.559429550316464,-0.561673578795992,-0.431884716383229,0.430159227344712],[0,0,0,0],[8.999999E+09,8.999999E+09,8.999999E+09,8.999999E+09,8.999999E+09,8.999999E+09]];
    LOCAL CONST Robtarget Tr_meulage_motif_1_122 := [[83.7916015625,-50.83070703125,66.95709375],[0.559429550316464,-0.561673578795992,-0.431884716383229,0.430159227344712],[0,0,0,0],[8.999999E+09,8.999999E+09,8.999999E+09,8.999999E+09,8.999999E+09,8.999999E+09]];
    LOCAL CONST Robtarget Tr_meulage_motif_1_123 := [[84.0464609375,-49.86373046875,66.95709375],[0.559429550316464,-0.561673578795992,-0.431884716383229,0.430159227344712],[0,0,0,0],[8.999999E+09,8.999999E+09,8.999999E+09,8.999999E+09,8.999999E+09,8.999999E+09]];
    LOCAL CONST Robtarget Tr_meulage_motif_1_124 := [[84.3013125,-48.89675,66.95709375],[0.559429550316464,-0.561673578795992,-0.431884716383229,0.430159227344712],[0,0,0,0],[8.999999E+09,8.999999E+09,8.999999E+09,8.999999E+09,8.999999E+09,8.999999E+09]];
    LOCAL CONST Robtarget Tr_meulage_motif_1_125 := [[84.5561640625,-47.92976953125,66.9571015625],[0.559429550316464,-0.561673578795992,-0.431884716383229,0.430159227344712],[0,0,0,0],[8.999999E+09,8.999999E+09,8.999999E+09,8.999999E+09,8.999999E+09,8.999999E+09]];
    LOCAL CONST Robtarget Tr_meulage_motif_1_126 := [[84.811015625,-46.9627890625,66.9571015625],[0.559429550316464,-0.561673578795992,-0.431884716383229,0.430159227344712],[0,0,0,0],[8.999999E+09,8.999999E+09,8.999999E+09,8.999999E+09,8.999999E+09,8.999999E+09]];
    LOCAL CONST Robtarget Tr_meulage_motif_1_127 := [[85.0658671875,-45.99580859375,66.9571015625],[0.559429550316464,-0.561673578795992,-0.431884716383229,0.430159227344712],[0,0,0,0],[8.999999E+09,8.999999E+09,8.999999E+09,8.999999E+09,8.999999E+09,8.999999E+09]];
    LOCAL CONST Robtarget Tr_meulage_motif_1_128 := [[85.3207265625,-45.02883203125,66.9571015625],[0.559429550316464,-0.561673578795992,-0.431884716383229,0.430159227344712],[0,0,0,0],[8.999999E+09,8.999999E+09,8.999999E+09,8.999999E+09,8.999999E+09,8.999999E+09]];
    LOCAL CONST Robtarget Tr_meulage_motif_1_129 := [[85.575578125,-44.0618515625,66.957109375],[0.559429550316464,-0.561673578795992,-0.431884716383229,0.430159227344712],[0,0,0,0],[8.999999E+09,8.999999E+09,8.999999E+09,8.999999E+09,8.999999E+09,8.999999E+09]];
    LOCAL CONST Robtarget Tr_meulage_motif_1_130 := [[85.8304296875,-43.09487109375,66.957109375],[0.559429550316464,-0.561673578795992,-0.431884716383229,0.430159227344712],[0,0,0,0],[8.999999E+09,8.999999E+09,8.999999E+09,8.999999E+09,8.999999E+09,8.999999E+09]];
    LOCAL CONST Robtarget Tr_meulage_motif_1_131 := [[86.08528125,-42.127890625,66.957109375],[0.559429550316464,-0.561673578795992,-0.431884716383229,0.430159227344712],[0,0,0,0],[8.999999E+09,8.999999E+09,8.999999E+09,8.999999E+09,8.999999E+09,8.999999E+09]];
    LOCAL CONST Robtarget Tr_meulage_motif_1_132 := [[86.340140625,-41.16091015625,66.957109375],[0.559429550316464,-0.561673578795992,-0.431884716383229,0.430159227344712],[0,0,0,0],[8.999999E+09,8.999999E+09,8.999999E+09,8.999999E+09,8.999999E+09,8.999999E+09]];
    LOCAL CONST Robtarget Tr_meulage_motif_1_133 := [[86.5949921875,-40.19393359375,66.9571171875],[0.559429550316464,-0.561673578795992,-0.431884716383229,0.430159227344712],[0,0,0,0],[8.999999E+09,8.999999E+09,8.999999E+09,8.999999E+09,8.999999E+09,8.999999E+09]];
    LOCAL CONST Robtarget Tr_meulage_motif_1_134 := [[86.84984375,-39.226953125,66.9571171875],[0.559429550316464,-0.561673578795992,-0.431884716383229,0.430159227344712],[0,0,0,0],[8.999999E+09,8.999999E+09,8.999999E+09,8.999999E+09,8.999999E+09,8.999999E+09]];
    LOCAL CONST Robtarget Tr_meulage_motif_1_135 := [[87.1046953125,-38.25997265625,66.9571171875],[0.559429550316464,-0.561673578795992,-0.431884716383229,0.430159227344712],[0,0,0,0],[8.999999E+09,8.999999E+09,8.999999E+09,8.999999E+09,8.999999E+09,8.999999E+09]];
    LOCAL CONST Robtarget Tr_meulage_motif_1_136 := [[87.3595546875,-37.2929921875,66.9571171875],[0.559429550316464,-0.561673578795992,-0.431884716383229,0.430159227344712],[0,0,0,0],[8.999999E+09,8.999999E+09,8.999999E+09,8.999999E+09,8.999999E+09,8.999999E+09]];
    LOCAL CONST Robtarget Tr_meulage_motif_1_137 := [[87.61440625,-36.32601171875,66.957125],[0.559429550316464,-0.561673578795992,-0.431884716383229,0.430159227344712],[0,0,0,0],[8.999999E+09,8.999999E+09,8.999999E+09,8.999999E+09,8.999999E+09,8.999999E+09]];
    LOCAL CONST Robtarget Tr_meulage_motif_1_138 := [[87.86709375,-35.36615234375,66.84653125],[0.559429550316464,-0.561673578795992,-0.431884716383229,0.430159227344712],[0,0,0,0],[8.999999E+09,8.999999E+09,8.999999E+09,8.999999E+09,8.999999E+09,8.999999E+09]];
    LOCAL CONST Robtarget Tr_meulage_motif_1_139 := [[88.107796875,-34.4507734375,66.63534375],[0.559429550316464,-0.561673578795992,-0.431884716383229,0.430159227344712],[0,0,0,0],[8.999999E+09,8.999999E+09,8.999999E+09,8.999999E+09,8.999999E+09,8.999999E+09]];
    LOCAL CONST Robtarget Tr_meulage_motif_1_140 := [[88.324453125,-33.62603515625,66.3635078125],[0.559429550316464,-0.561673578795992,-0.431884716383229,0.430159227344712],[0,0,0,0],[8.999999E+09,8.999999E+09,8.999999E+09,8.999999E+09,8.999999E+09,8.999999E+09]];
    LOCAL CONST Robtarget Tr_meulage_motif_1_141 := [[88.51490625,-32.90068359375,66.0875703125],[0.559429550316464,-0.561673578795992,-0.431884716383229,0.430159227344712],[0,0,0,0],[8.999999E+09,8.999999E+09,8.999999E+09,8.999999E+09,8.999999E+09,8.999999E+09]];
    LOCAL CONST Robtarget Tr_meulage_motif_1_142 := [[88.794015625,-31.83558203125,65.47144921875],[0.559429550316464,-0.561673578795992,-0.431884716383229,0.430159227344712],[0,0,0,0],[8.999999E+09,8.999999E+09,8.999999E+09,8.999999E+09,8.999999E+09,8.999999E+09]];
    LOCAL CONST Robtarget Tr_meulage_motif_1_143 := [[89.052890625,-30.84496875,64.623796875],[0.559429550316464,-0.561673578795992,-0.431884716383229,0.430159227344712],[0,0,0,0],[8.999999E+09,8.999999E+09,8.999999E+09,8.999999E+09,8.999999E+09,8.999999E+09]];
    LOCAL CONST Robtarget Tr_meulage_motif_1_144 := [[89.2664296875,-30.02464453125,63.59992578125],[0.559429550316464,-0.561673578795992,-0.431884716383229,0.430159227344712],[0,0,0,0],[8.999999E+09,8.999999E+09,8.999999E+09,8.999999E+09,8.999999E+09,8.999999E+09]];
    LOCAL CONST Robtarget Tr_meulage_motif_1_145 := [[89.3881171875,-29.551888671875,62.48374609375],[0.559429550316464,-0.561673578795992,-0.431884716383229,0.430159227344712],[0,0,0,0],[8.999999E+09,8.999999E+09,8.999999E+09,8.999999E+09,8.999999E+09,8.999999E+09]];
    LOCAL CONST Robtarget Tr_meulage_motif_1_146 := [[89.3933203125,-29.525271484375,61.78777734375],[0.559429550316464,-0.561673578795992,-0.431884716383229,0.430159227344712],[0,0,0,0],[8.999999E+09,8.999999E+09,8.999999E+09,8.999999E+09,8.999999E+09,8.999999E+09]];
    LOCAL CONST Robtarget Tr_meulage_motif_1_147 := [[89.3917109375,-29.524845703125,61.12653125],[0.559429550316464,-0.561673578795992,-0.431884716383229,0.430159227344712],[0,0,0,0],[8.999999E+09,8.999999E+09,8.999999E+09,8.999999E+09,8.999999E+09,8.999999E+09]];
    LOCAL CONST Robtarget Tr_meulage_motif_1_148 := [[89.3761171875,-29.577484375,60.4654375],[0.559429550316464,-0.561673578795992,-0.431884716383229,0.430159227344712],[0,0,0,0],[8.999999E+09,8.999999E+09,8.999999E+09,8.999999E+09,8.999999E+09,8.999999E+09]];
    LOCAL CONST Robtarget Tr_meulage_motif_1_149 := [[89.2464609375,-30.05854296875,59.36369140625],[0.559429550316464,-0.561673578795992,-0.431884716383229,0.430159227344712],[0,0,0,0],[8.999999E+09,8.999999E+09,8.999999E+09,8.999999E+09,8.999999E+09,8.999999E+09]];
    LOCAL CONST Robtarget Tr_meulage_motif_1_150 := [[89.0256953125,-30.886234375,58.35706640625],[0.559429550316464,-0.561673578795992,-0.431884716383229,0.430159227344712],[0,0,0,0],[8.999999E+09,8.999999E+09,8.999999E+09,8.999999E+09,8.999999E+09,8.999999E+09]];
    LOCAL CONST Robtarget Tr_meulage_motif_1_151 := [[88.762859375,-31.8753125,57.52819140625],[0.559429550316464,-0.561673578795992,-0.431884716383229,0.430159227344712],[0,0,0,0],[8.999999E+09,8.999999E+09,8.999999E+09,8.999999E+09,8.999999E+09,8.999999E+09]];
    LOCAL CONST Robtarget Tr_meulage_motif_1_152 := [[88.5867890625,-32.53946484375,57.13244140625],[0.559429550316464,-0.561673578795992,-0.431884716383229,0.430159227344712],[0,0,0,0],[8.999999E+09,8.999999E+09,8.999999E+09,8.999999E+09,8.999999E+09,8.999999E+09]];
    LOCAL CONST Robtarget Tr_meulage_motif_1_153 := [[88.2904453125,-33.6590625,56.64491015625],[0.559429550316464,-0.561673578795992,-0.431884716383229,0.430159227344712],[0,0,0,0],[8.999999E+09,8.999999E+09,8.999999E+09,8.999999E+09,8.999999E+09,8.999999E+09]];
    LOCAL CONST Robtarget Tr_meulage_motif_1_154 := [[88.0744453125,-34.4760234375,56.38081640625],[0.559429550316464,-0.561673578795992,-0.431884716383229,0.430159227344712],[0,0,0,0],[8.999999E+09,8.999999E+09,8.999999E+09,8.999999E+09,8.999999E+09,8.999999E+09]];
    LOCAL CONST Robtarget Tr_meulage_motif_1_155 := [[87.836421875,-35.3771171875,56.17634765625],[0.559429550316464,-0.561673578795992,-0.431884716383229,0.430159227344712],[0,0,0,0],[8.999999E+09,8.999999E+09,8.999999E+09,8.999999E+09,8.999999E+09,8.999999E+09]];
    LOCAL CONST Robtarget Tr_meulage_motif_1_156 := [[87.586,-36.3261953125,56.06775],[0.559429550316464,-0.561673578795992,-0.431884716383229,0.430159227344712],[0,0,0,0],[8.999999E+09,8.999999E+09,8.999999E+09,8.999999E+09,8.999999E+09,8.999999E+09]];
    LOCAL CONST Robtarget Tr_meulage_motif_1_157 := [[87.3327734375,-37.2859140625,55.95715625],[0.559429550316464,-0.561673578795992,-0.431884716383229,0.430159227344712],[0,0,0,0],[8.999999E+09,8.999999E+09,8.999999E+09,8.999999E+09,8.999999E+09,8.999999E+09]];
    LOCAL CONST Robtarget Tr_meulage_motif_1_158 := [[87.077921875,-38.25289453125,55.95715234375],[0.559429550316464,-0.561673578795992,-0.431884716383229,0.430159227344712],[0,0,0,0],[8.999999E+09,8.999999E+09,8.999999E+09,8.999999E+09,8.999999E+09,8.999999E+09]];
    LOCAL CONST Robtarget Tr_meulage_motif_1_159 := [[86.8230703125,-39.21987109375,55.95715234375],[0.559429550316464,-0.561673578795992,-0.431884716383229,0.430159227344712],[0,0,0,0],[8.999999E+09,8.999999E+09,8.999999E+09,8.999999E+09,8.999999E+09,8.999999E+09]];
    LOCAL CONST Robtarget Tr_meulage_motif_1_160 := [[86.5682109375,-40.1868515625,55.9571484375],[0.559429550316464,-0.561673578795992,-0.431884716383229,0.430159227344712],[0,0,0,0],[8.999999E+09,8.999999E+09,8.999999E+09,8.999999E+09,8.999999E+09,8.999999E+09]];
    LOCAL CONST Robtarget Tr_meulage_motif_1_161 := [[86.313359375,-41.15383203125,55.9571484375],[0.559429550316464,-0.561673578795992,-0.431884716383229,0.430159227344712],[0,0,0,0],[8.999999E+09,8.999999E+09,8.999999E+09,8.999999E+09,8.999999E+09,8.999999E+09]];
    LOCAL CONST Robtarget Tr_meulage_motif_1_162 := [[86.0585078125,-42.1208125,55.95714453125],[0.559429550316464,-0.561673578795992,-0.431884716383229,0.430159227344712],[0,0,0,0],[8.999999E+09,8.999999E+09,8.999999E+09,8.999999E+09,8.999999E+09,8.999999E+09]];
    LOCAL CONST Robtarget Tr_meulage_motif_1_163 := [[85.80365625,-43.08779296875,55.95714453125],[0.559429550316464,-0.561673578795992,-0.431884716383229,0.430159227344712],[0,0,0,0],[8.999999E+09,8.999999E+09,8.999999E+09,8.999999E+09,8.999999E+09,8.999999E+09]];
    LOCAL CONST Robtarget Tr_meulage_motif_1_164 := [[85.548796875,-44.05476953125,55.957140625],[0.559429550316464,-0.561673578795992,-0.431884716383229,0.430159227344712],[0,0,0,0],[8.999999E+09,8.999999E+09,8.999999E+09,8.999999E+09,8.999999E+09,8.999999E+09]];
    LOCAL CONST Robtarget Tr_meulage_motif_1_165 := [[85.2939453125,-45.02175,55.957140625],[0.559429550316464,-0.561673578795992,-0.431884716383229,0.430159227344712],[0,0,0,0],[8.999999E+09,8.999999E+09,8.999999E+09,8.999999E+09,8.999999E+09,8.999999E+09]];
    LOCAL CONST Robtarget Tr_meulage_motif_1_166 := [[85.03909375,-45.98873046875,55.95713671875],[0.559429550316464,-0.561673578795992,-0.431884716383229,0.430159227344712],[0,0,0,0],[8.999999E+09,8.999999E+09,8.999999E+09,8.999999E+09,8.999999E+09,8.999999E+09]];
    LOCAL CONST Robtarget Tr_meulage_motif_1_167 := [[84.7842421875,-46.9557109375,55.95713671875],[0.559429550316464,-0.561673578795992,-0.431884716383229,0.430159227344712],[0,0,0,0],[8.999999E+09,8.999999E+09,8.999999E+09,8.999999E+09,8.999999E+09,8.999999E+09]];
    LOCAL CONST Robtarget Tr_meulage_motif_1_168 := [[84.5293828125,-47.92269140625,55.9571328125],[0.559429550316464,-0.561673578795992,-0.431884716383229,0.430159227344712],[0,0,0,0],[8.999999E+09,8.999999E+09,8.999999E+09,8.999999E+09,8.999999E+09,8.999999E+09]];
    LOCAL CONST Robtarget Tr_meulage_motif_1_169 := [[84.27453125,-48.88966796875,55.9571328125],[0.559429550316464,-0.561673578795992,-0.431884716383229,0.430159227344712],[0,0,0,0],[8.999999E+09,8.999999E+09,8.999999E+09,8.999999E+09,8.999999E+09,8.999999E+09]];
    LOCAL CONST Robtarget Tr_meulage_motif_1_170 := [[84.0196796875,-49.8566484375,55.95712890625],[0.559429550316464,-0.561673578795992,-0.431884716383229,0.430159227344712],[0,0,0,0],[8.999999E+09,8.999999E+09,8.999999E+09,8.999999E+09,8.999999E+09,8.999999E+09]];
    LOCAL CONST Robtarget Tr_meulage_motif_1_171 := [[83.764828125,-50.82362890625,55.95712890625],[0.559429550316464,-0.561673578795992,-0.431884716383229,0.430159227344712],[0,0,0,0],[8.999999E+09,8.999999E+09,8.999999E+09,8.999999E+09,8.999999E+09,8.999999E+09]];
    LOCAL CONST Robtarget Tr_meulage_motif_1_172 := [[83.5099765625,-51.790609375,55.957125],[0.559429550316464,-0.561673578795992,-0.431884716383229,0.430159227344712],[0,0,0,0],[8.999999E+09,8.999999E+09,8.999999E+09,8.999999E+09,8.999999E+09,8.999999E+09]];
    LOCAL CONST Robtarget Tr_meulage_motif_1_173 := [[83.2551171875,-52.75758984375,55.957125],[0.559429550316464,-0.561673578795992,-0.431884716383229,0.430159227344712],[0,0,0,0],[8.999999E+09,8.999999E+09,8.999999E+09,8.999999E+09,8.999999E+09,8.999999E+09]];
    LOCAL CONST Robtarget Tr_meulage_motif_1_174 := [[83.000265625,-53.72456640625,55.95712109375],[0.559429550316464,-0.561673578795992,-0.431884716383229,0.430159227344712],[0,0,0,0],[8.999999E+09,8.999999E+09,8.999999E+09,8.999999E+09,8.999999E+09,8.999999E+09]];
    LOCAL CONST Robtarget Tr_meulage_motif_1_175 := [[82.7454140625,-54.691546875,55.95712109375],[0.559429550316464,-0.561673578795992,-0.431884716383229,0.430159227344712],[0,0,0,0],[8.999999E+09,8.999999E+09,8.999999E+09,8.999999E+09,8.999999E+09,8.999999E+09]];
    LOCAL CONST Robtarget Tr_meulage_motif_1_176 := [[82.4905625,-55.65852734375,55.9571171875],[0.559429550316464,-0.561673578795992,-0.431884716383229,0.430159227344712],[0,0,0,0],[8.999999E+09,8.999999E+09,8.999999E+09,8.999999E+09,8.999999E+09,8.999999E+09]];
    LOCAL CONST Robtarget Tr_meulage_motif_1_177 := [[82.235703125,-56.6255078125,55.9571171875],[0.559429550316464,-0.561673578795992,-0.431884716383229,0.430159227344712],[0,0,0,0],[8.999999E+09,8.999999E+09,8.999999E+09,8.999999E+09,8.999999E+09,8.999999E+09]];
    LOCAL CONST Robtarget Tr_meulage_motif_1_178 := [[81.9808515625,-57.59248828125,55.95711328125],[0.559429550316464,-0.561673578795992,-0.431884716383229,0.430159227344712],[0,0,0,0],[8.999999E+09,8.999999E+09,8.999999E+09,8.999999E+09,8.999999E+09,8.999999E+09]];
    LOCAL CONST Robtarget Tr_meulage_motif_1_179 := [[81.726,-58.55946484375,55.95711328125],[0.559429550316464,-0.561673578795992,-0.431884716383229,0.430159227344712],[0,0,0,0],[8.999999E+09,8.999999E+09,8.999999E+09,8.999999E+09,8.999999E+09,8.999999E+09]];
    LOCAL CONST Robtarget Tr_meulage_motif_1_180 := [[81.4711484375,-59.5264453125,55.957109375],[0.559429550316464,-0.561673578795992,-0.431884716383229,0.430159227344712],[0,0,0,0],[8.999999E+09,8.999999E+09,8.999999E+09,8.999999E+09,8.999999E+09,8.999999E+09]];
    LOCAL CONST Robtarget Tr_meulage_motif_1_181 := [[81.2162890625,-60.49342578125,55.957109375],[0.559429550316464,-0.561673578795992,-0.431884716383229,0.430159227344712],[0,0,0,0],[8.999999E+09,8.999999E+09,8.999999E+09,8.999999E+09,8.999999E+09,8.999999E+09]];
    LOCAL CONST Robtarget Tr_meulage_motif_1_182 := [[80.9614375,-61.46040625,55.95710546875],[0.559429550316464,-0.561673578795992,-0.431884716383229,0.430159227344712],[0,0,0,0],[8.999999E+09,8.999999E+09,8.999999E+09,8.999999E+09,8.999999E+09,8.999999E+09]];
    LOCAL CONST Robtarget Tr_meulage_motif_1_183 := [[80.7065859375,-62.42738671875,55.95710546875],[0.559429550316464,-0.561673578795992,-0.431884716383229,0.430159227344712],[0,0,0,0],[8.999999E+09,8.999999E+09,8.999999E+09,8.999999E+09,8.999999E+09,8.999999E+09]];
    LOCAL CONST Robtarget Tr_meulage_motif_1_184 := [[80.451734375,-63.39436328125,55.9571015625],[0.559429550316464,-0.561673578795992,-0.431884716383229,0.430159227344712],[0,0,0,0],[8.999999E+09,8.999999E+09,8.999999E+09,8.999999E+09,8.999999E+09,8.999999E+09]];
    LOCAL CONST Robtarget Tr_meulage_motif_1_185 := [[80.196875,-64.36134375,55.9571015625],[0.559429550316464,-0.561673578795992,-0.431884716383229,0.430159227344712],[0,0,0,0],[8.999999E+09,8.999999E+09,8.999999E+09,8.999999E+09,8.999999E+09,8.999999E+09]];
    LOCAL CONST Robtarget Tr_meulage_motif_1_186 := [[79.9420234375,-65.32832421875,55.95709765625],[0.559429550316464,-0.561673578795992,-0.431884716383229,0.430159227344712],[0,0,0,0],[8.999999E+09,8.999999E+09,8.999999E+09,8.999999E+09,8.999999E+09,8.999999E+09]];
    LOCAL CONST Robtarget Tr_meulage_motif_1_187 := [[79.687171875,-66.2953046875,55.95709765625],[0.559429550316464,-0.561673578795992,-0.431884716383229,0.430159227344712],[0,0,0,0],[8.999999E+09,8.999999E+09,8.999999E+09,8.999999E+09,8.999999E+09,8.999999E+09]];
    LOCAL CONST Robtarget Tr_meulage_motif_1_188 := [[79.4339453125,-67.2550234375,55.84650390625],[0.559429550316464,-0.561673578795992,-0.431884716383229,0.430159227344712],[0,0,0,0],[8.999999E+09,8.999999E+09,8.999999E+09,8.999999E+09,8.999999E+09,8.999999E+09]];
    LOCAL CONST Robtarget Tr_meulage_motif_1_189 := [[79.1922109375,-68.1701328125,55.6353125],[0.559429550316464,-0.561673578795992,-0.431884716383229,0.430159227344712],[0,0,0,0],[8.999999E+09,8.999999E+09,8.999999E+09,8.999999E+09,8.999999E+09,8.999999E+09]];
    LOCAL CONST Robtarget Tr_meulage_motif_1_190 := [[78.974234375,-68.994515625,55.36346875],[0.559429550316464,-0.561673578795992,-0.431884716383229,0.430159227344712],[0,0,0,0],[8.999999E+09,8.999999E+09,8.999999E+09,8.999999E+09,8.999999E+09,8.999999E+09]];
    LOCAL CONST Robtarget Tr_meulage_motif_1_191 := [[78.7921640625,-69.682328125,55.059328125],[0.559429550316464,-0.561673578795992,-0.431884716383229,0.430159227344712],[0,0,0,0],[8.999999E+09,8.999999E+09,8.999999E+09,8.999999E+09,8.999999E+09,8.999999E+09]];
    LOCAL CONST Robtarget Tr_meulage_motif_1_192 := [[78.5269140625,-70.6822109375,54.396796875],[0.559429550316464,-0.561673578795992,-0.431884716383229,0.430159227344712],[0,0,0,0],[8.999999E+09,8.999999E+09,8.999999E+09,8.999999E+09,8.999999E+09,8.999999E+09]];
    LOCAL CONST Robtarget Tr_meulage_motif_1_193 := [[78.2948515625,-71.5537890625,53.49484375],[0.559429550316464,-0.561673578795992,-0.431884716383229,0.430159227344712],[0,0,0,0],[8.999999E+09,8.999999E+09,8.999999E+09,8.999999E+09,8.999999E+09,8.999999E+09]];
    LOCAL CONST Robtarget Tr_meulage_motif_1_194 := [[78.15596875,-72.0704140625,52.44883203125],[0.559429550316464,-0.561673578795992,-0.431884716383229,0.430159227344712],[0,0,0,0],[8.999999E+09,8.999999E+09,8.999999E+09,8.999999E+09,8.999999E+09,8.999999E+09]];
    LOCAL CONST Robtarget Tr_meulage_motif_1_195 := [[78.1071875,-72.2486484375,51.75559765625],[0.559429550316464,-0.561673578795992,-0.431884716383229,0.430159227344712],[0,0,0,0],[8.999999E+09,8.999999E+09,8.999999E+09,8.999999E+09,8.999999E+09,8.999999E+09]];
    LOCAL CONST Robtarget Tr_meulage_motif_1_196 := [[78.089046875,-72.309890625,50.9856015625],[0.559429550316464,-0.561673578795992,-0.431884716383229,0.430159227344712],[0,0,0,0],[8.999999E+09,8.999999E+09,8.999999E+09,8.999999E+09,8.999999E+09,8.999999E+09]];
    LOCAL CONST Robtarget Tr_meulage_motif_1_197 := [[78.1042265625,-72.244671875,50.21574609375],[0.559429550316464,-0.561673578795992,-0.431884716383229,0.430159227344712],[0,0,0,0],[8.999999E+09,8.999999E+09,8.999999E+09,8.999999E+09,8.999999E+09,8.999999E+09]];
    LOCAL CONST Robtarget Tr_meulage_motif_1_198 := [[78.20846875,-71.83821875,49.1075],[0.559429550316464,-0.561673578795992,-0.431884716383229,0.430159227344712],[0,0,0,0],[8.999999E+09,8.999999E+09,8.999999E+09,8.999999E+09,8.999999E+09,8.999999E+09]];
    LOCAL CONST Robtarget Tr_meulage_motif_1_199 := [[78.3126328125,-71.4372109375,48.5218125],[0.559429550316464,-0.561673578795992,-0.431884716383229,0.430159227344712],[0,0,0,0],[8.999999E+09,8.999999E+09,8.999999E+09,8.999999E+09,8.999999E+09,8.999999E+09]];
    LOCAL CONST Robtarget Tr_meulage_motif_1_200 := [[78.5365546875,-70.5788046875,47.6346640625],[0.559429550316464,-0.561673578795992,-0.431884716383229,0.430159227344712],[0,0,0,0],[8.999999E+09,8.999999E+09,8.999999E+09,8.999999E+09,8.999999E+09,8.999999E+09]];
    LOCAL CONST Robtarget Tr_meulage_motif_1_201 := [[78.6848125,-70.0121875,47.2203828125],[0.559429550316464,-0.561673578795992,-0.431884716383229,0.430159227344712],[0,0,0,0],[8.999999E+09,8.999999E+09,8.999999E+09,8.999999E+09,8.999999E+09,8.999999E+09]];
    LOCAL CONST Robtarget Tr_meulage_motif_1_202 := [[78.968390625,-68.93084375,46.67626171875],[0.559429550316464,-0.561673578795992,-0.431884716383229,0.430159227344712],[0,0,0,0],[8.999999E+09,8.999999E+09,8.999999E+09,8.999999E+09,8.999999E+09,8.999999E+09]];
    LOCAL CONST Robtarget Tr_meulage_motif_1_203 := [[79.178078125,-68.132328125,46.380765625],[0.559429550316464,-0.561673578795992,-0.431884716383229,0.430159227344712],[0,0,0,0],[8.999999E+09,8.999999E+09,8.999999E+09,8.999999E+09,8.999999E+09,8.999999E+09]];
    LOCAL CONST Robtarget Tr_meulage_motif_1_204 := [[79.4151015625,-67.23096875,46.17628125],[0.559429550316464,-0.561673578795992,-0.431884716383229,0.430159227344712],[0,0,0,0],[8.999999E+09,8.999999E+09,8.999999E+09,8.999999E+09,8.999999E+09,8.999999E+09]];
    LOCAL CONST Robtarget Tr_meulage_motif_1_205 := [[79.6649921875,-66.28175,46.06773828125],[0.559429550316464,-0.561673578795992,-0.431884716383229,0.430159227344712],[0,0,0,0],[8.999999E+09,8.999999E+09,8.999999E+09,8.999999E+09,8.999999E+09,8.999999E+09]];
    LOCAL CONST Robtarget Tr_meulage_motif_1_206 := [[79.9176796875,-65.32188671875,45.9571328125],[0.559429550316464,-0.561673578795992,-0.431884716383229,0.430159227344712],[0,0,0,0],[8.999999E+09,8.999999E+09,8.999999E+09,8.999999E+09,8.999999E+09,8.999999E+09]];
    LOCAL CONST Robtarget Tr_meulage_motif_1_207 := [[80.1725390625,-64.35491015625,45.9571328125],[0.559429550316464,-0.561673578795992,-0.431884716383229,0.430159227344712],[0,0,0,0],[8.999999E+09,8.999999E+09,8.999999E+09,8.999999E+09,8.999999E+09,8.999999E+09]];
    LOCAL CONST Robtarget Tr_meulage_motif_1_208 := [[80.427390625,-63.3879296875,45.95713671875],[0.559429550316464,-0.561673578795992,-0.431884716383229,0.430159227344712],[0,0,0,0],[8.999999E+09,8.999999E+09,8.999999E+09,8.999999E+09,8.999999E+09,8.999999E+09]];
    LOCAL CONST Robtarget Tr_meulage_motif_1_209 := [[80.6822421875,-62.42094921875,45.95713671875],[0.559429550316464,-0.561673578795992,-0.431884716383229,0.430159227344712],[0,0,0,0],[8.999999E+09,8.999999E+09,8.999999E+09,8.999999E+09,8.999999E+09,8.999999E+09]];
    LOCAL CONST Robtarget Tr_meulage_motif_1_210 := [[80.93709375,-61.45396875,45.957140625],[0.559429550316464,-0.561673578795992,-0.431884716383229,0.430159227344712],[0,0,0,0],[8.999999E+09,8.999999E+09,8.999999E+09,8.999999E+09,8.999999E+09,8.999999E+09]];
    LOCAL CONST Robtarget Tr_meulage_motif_1_211 := [[81.1919453125,-60.48698828125,45.957140625],[0.559429550316464,-0.561673578795992,-0.431884716383229,0.430159227344712],[0,0,0,0],[8.999999E+09,8.999999E+09,8.999999E+09,8.999999E+09,8.999999E+09,8.999999E+09]];
    LOCAL CONST Robtarget Tr_meulage_motif_1_212 := [[81.4468046875,-59.52001171875,45.95714453125],[0.559429550316464,-0.561673578795992,-0.431884716383229,0.430159227344712],[0,0,0,0],[8.999999E+09,8.999999E+09,8.999999E+09,8.999999E+09,8.999999E+09,8.999999E+09]];
    LOCAL CONST Robtarget Tr_meulage_motif_1_213 := [[81.70165625,-58.55303125,45.95714453125],[0.559429550316464,-0.561673578795992,-0.431884716383229,0.430159227344712],[0,0,0,0],[8.999999E+09,8.999999E+09,8.999999E+09,8.999999E+09,8.999999E+09,8.999999E+09]];
    LOCAL CONST Robtarget Tr_meulage_motif_1_214 := [[81.9565078125,-57.58605078125,45.9571484375],[0.559429550316464,-0.561673578795992,-0.431884716383229,0.430159227344712],[0,0,0,0],[8.999999E+09,8.999999E+09,8.999999E+09,8.999999E+09,8.999999E+09,8.999999E+09]];
    LOCAL CONST Robtarget Tr_meulage_motif_1_215 := [[82.211359375,-56.6190703125,45.9571484375],[0.559429550316464,-0.561673578795992,-0.431884716383229,0.430159227344712],[0,0,0,0],[8.999999E+09,8.999999E+09,8.999999E+09,8.999999E+09,8.999999E+09,8.999999E+09]];
    LOCAL CONST Robtarget Tr_meulage_motif_1_216 := [[82.46621875,-55.65208984375,45.95715234375],[0.559429550316464,-0.561673578795992,-0.431884716383229,0.430159227344712],[0,0,0,0],[8.999999E+09,8.999999E+09,8.999999E+09,8.999999E+09,8.999999E+09,8.999999E+09]];
    LOCAL CONST Robtarget Tr_meulage_motif_1_217 := [[82.7210703125,-54.68511328125,45.95715234375],[0.559429550316464,-0.561673578795992,-0.431884716383229,0.430159227344712],[0,0,0,0],[8.999999E+09,8.999999E+09,8.999999E+09,8.999999E+09,8.999999E+09,8.999999E+09]];
    LOCAL CONST Robtarget Tr_meulage_motif_1_218 := [[82.975921875,-53.7181328125,45.95715625],[0.559429550316464,-0.561673578795992,-0.431884716383229,0.430159227344712],[0,0,0,0],[8.999999E+09,8.999999E+09,8.999999E+09,8.999999E+09,8.999999E+09,8.999999E+09]];
    LOCAL CONST Robtarget Tr_meulage_motif_1_219 := [[83.2307734375,-52.75115234375,45.95715625],[0.559429550316464,-0.561673578795992,-0.431884716383229,0.430159227344712],[0,0,0,0],[8.999999E+09,8.999999E+09,8.999999E+09,8.999999E+09,8.999999E+09,8.999999E+09]];
    LOCAL CONST Robtarget Tr_meulage_motif_1_220 := [[83.4856328125,-51.784171875,45.95716015625],[0.559429550316464,-0.561673578795992,-0.431884716383229,0.430159227344712],[0,0,0,0],[8.999999E+09,8.999999E+09,8.999999E+09,8.999999E+09,8.999999E+09,8.999999E+09]];
    LOCAL CONST Robtarget Tr_meulage_motif_1_221 := [[83.740484375,-50.81719140625,45.95716015625],[0.559429550316464,-0.561673578795992,-0.431884716383229,0.430159227344712],[0,0,0,0],[8.999999E+09,8.999999E+09,8.999999E+09,8.999999E+09,8.999999E+09,8.999999E+09]];
    LOCAL CONST Robtarget Tr_meulage_motif_1_222 := [[83.9953359375,-49.85021484375,45.9571640625],[0.559429550316464,-0.561673578795992,-0.431884716383229,0.430159227344712],[0,0,0,0],[8.999999E+09,8.999999E+09,8.999999E+09,8.999999E+09,8.999999E+09,8.999999E+09]];
    LOCAL CONST Robtarget Tr_meulage_motif_1_223 := [[84.2501875,-48.883234375,45.9571640625],[0.559429550316464,-0.561673578795992,-0.431884716383229,0.430159227344712],[0,0,0,0],[8.999999E+09,8.999999E+09,8.999999E+09,8.999999E+09,8.999999E+09,8.999999E+09]];
    LOCAL CONST Robtarget Tr_meulage_motif_1_224 := [[84.505046875,-47.91625390625,45.95716796875],[0.559429550316464,-0.561673578795992,-0.431884716383229,0.430159227344712],[0,0,0,0],[8.999999E+09,8.999999E+09,8.999999E+09,8.999999E+09,8.999999E+09,8.999999E+09]];
    LOCAL CONST Robtarget Tr_meulage_motif_1_225 := [[84.7598984375,-46.9492734375,45.95716796875],[0.559429550316464,-0.561673578795992,-0.431884716383229,0.430159227344712],[0,0,0,0],[8.999999E+09,8.999999E+09,8.999999E+09,8.999999E+09,8.999999E+09,8.999999E+09]];
    LOCAL CONST Robtarget Tr_meulage_motif_1_226 := [[85.01475,-45.98229296875,45.957171875],[0.559429550316464,-0.561673578795992,-0.431884716383229,0.430159227344712],[0,0,0,0],[8.999999E+09,8.999999E+09,8.999999E+09,8.999999E+09,8.999999E+09,8.999999E+09]];
    LOCAL CONST Robtarget Tr_meulage_motif_1_227 := [[85.2696015625,-45.01531640625,45.957171875],[0.559429550316464,-0.561673578795992,-0.431884716383229,0.430159227344712],[0,0,0,0],[8.999999E+09,8.999999E+09,8.999999E+09,8.999999E+09,8.999999E+09,8.999999E+09]];
    LOCAL CONST Robtarget Tr_meulage_motif_1_228 := [[85.5244609375,-44.0483359375,45.95717578125],[0.559429550316464,-0.561673578795992,-0.431884716383229,0.430159227344712],[0,0,0,0],[8.999999E+09,8.999999E+09,8.999999E+09,8.999999E+09,8.999999E+09,8.999999E+09]];
    LOCAL CONST Robtarget Tr_meulage_motif_1_229 := [[85.7793125,-43.08135546875,45.95717578125],[0.559429550316464,-0.561673578795992,-0.431884716383229,0.430159227344712],[0,0,0,0],[8.999999E+09,8.999999E+09,8.999999E+09,8.999999E+09,8.999999E+09,8.999999E+09]];
    LOCAL CONST Robtarget Tr_meulage_motif_1_230 := [[86.0341640625,-42.114375,45.9571796875],[0.559429550316464,-0.561673578795992,-0.431884716383229,0.430159227344712],[0,0,0,0],[8.999999E+09,8.999999E+09,8.999999E+09,8.999999E+09,8.999999E+09,8.999999E+09]];
    LOCAL CONST Robtarget Tr_meulage_motif_1_231 := [[86.289015625,-41.14739453125,45.9571796875],[0.559429550316464,-0.561673578795992,-0.431884716383229,0.430159227344712],[0,0,0,0],[8.999999E+09,8.999999E+09,8.999999E+09,8.999999E+09,8.999999E+09,8.999999E+09]];
    LOCAL CONST Robtarget Tr_meulage_motif_1_232 := [[86.5438671875,-40.18041796875,45.95718359375],[0.559429550316464,-0.561673578795992,-0.431884716383229,0.430159227344712],[0,0,0,0],[8.999999E+09,8.999999E+09,8.999999E+09,8.999999E+09,8.999999E+09,8.999999E+09]];
    LOCAL CONST Robtarget Tr_meulage_motif_1_233 := [[86.7987265625,-39.2134375,45.95718359375],[0.559429550316464,-0.561673578795992,-0.431884716383229,0.430159227344712],[0,0,0,0],[8.999999E+09,8.999999E+09,8.999999E+09,8.999999E+09,8.999999E+09,8.999999E+09]];
    LOCAL CONST Robtarget Tr_meulage_motif_1_234 := [[87.053578125,-38.24645703125,45.9571875],[0.559429550316464,-0.561673578795992,-0.431884716383229,0.430159227344712],[0,0,0,0],[8.999999E+09,8.999999E+09,8.999999E+09,8.999999E+09,8.999999E+09,8.999999E+09]];
    LOCAL CONST Robtarget Tr_meulage_motif_1_235 := [[87.3084296875,-37.2794765625,45.9571875],[0.559429550316464,-0.561673578795992,-0.431884716383229,0.430159227344712],[0,0,0,0],[8.999999E+09,8.999999E+09,8.999999E+09,8.999999E+09,8.999999E+09,8.999999E+09]];
    LOCAL CONST Robtarget Tr_meulage_motif_1_236 := [[87.56328125,-36.31249609375,45.9571875],[0.559429550316464,-0.561673578795992,-0.431884716383229,0.430159227344712],[0,0,0,0],[8.999999E+09,8.999999E+09,8.999999E+09,8.999999E+09,8.999999E+09,8.999999E+09]];
    LOCAL CONST Robtarget Tr_meulage_motif_1_237 := [[87.8159765625,-35.35263671875,45.84658203125],[0.559429550316464,-0.561673578795992,-0.431884716383229,0.430159227344712],[0,0,0,0],[8.999999E+09,8.999999E+09,8.999999E+09,8.999999E+09,8.999999E+09,8.999999E+09]];
    LOCAL CONST Robtarget Tr_meulage_motif_1_238 := [[88.0566796875,-34.4372578125,45.6353984375],[0.559429550316464,-0.561673578795992,-0.431884716383229,0.430159227344712],[0,0,0,0],[8.999999E+09,8.999999E+09,8.999999E+09,8.999999E+09,8.999999E+09,8.999999E+09]];
    LOCAL CONST Robtarget Tr_meulage_motif_1_239 := [[88.2733359375,-33.61251953125,45.3635703125],[0.559429550316464,-0.561673578795992,-0.431884716383229,0.430159227344712],[0,0,0,0],[8.999999E+09,8.999999E+09,8.999999E+09,8.999999E+09,8.999999E+09,8.999999E+09]];
    LOCAL CONST Robtarget Tr_meulage_motif_1_240 := [[88.453921875,-32.92431640625,45.05943359375],[0.559429550316464,-0.561673578795992,-0.431884716383229,0.430159227344712],[0,0,0,0],[8.999999E+09,8.999999E+09,8.999999E+09,8.999999E+09,8.999999E+09,8.999999E+09]];
    LOCAL CONST Robtarget Tr_meulage_motif_1_241 := [[88.7159453125,-31.92358203125,44.39690625],[0.559429550316464,-0.561673578795992,-0.431884716383229,0.430159227344712],[0,0,0,0],[8.999999E+09,8.999999E+09,8.999999E+09,8.999999E+09,8.999999E+09,8.999999E+09]];
    LOCAL CONST Robtarget Tr_meulage_motif_1_242 := [[88.9208203125,-31.136943359375,43.45712890625],[0.559429550316464,-0.561673578795992,-0.431884716383229,0.430159227344712],[0,0,0,0],[8.999999E+09,8.999999E+09,8.999999E+09,8.999999E+09,8.999999E+09,8.999999E+09]];
    LOCAL CONST Robtarget Tr_meulage_motif_1_243 := [[89.00821875,-30.795501953125,42.4607734375],[0.559429550316464,-0.561673578795992,-0.431884716383229,0.430159227344712],[0,0,0,0],[8.999999E+09,8.999999E+09,8.999999E+09,8.999999E+09,8.999999E+09,8.999999E+09]];
    LOCAL CONST Robtarget Tr_meulage_motif_1_244 := [[88.9993046875,-30.8238203125,41.90323046875],[0.559429550316464,-0.561673578795992,-0.431884716383229,0.430159227344712],[0,0,0,0],[8.999999E+09,8.999999E+09,8.999999E+09,8.999999E+09,8.999999E+09,8.999999E+09]];
    LOCAL CONST Robtarget Tr_meulage_motif_1_245 := [[88.9993828125,-30.819380859375,41.48532421875],[0.559429550316464,-0.561673578795992,-0.431884716383229,0.430159227344712],[0,0,0,0],[8.999999E+09,8.999999E+09,8.999999E+09,8.999999E+09,8.999999E+09,8.999999E+09]];
    LOCAL CONST Robtarget Tr_meulage_motif_1_246 := [[88.9047265625,-31.168955078125,40.516],[0.559429550316464,-0.561673578795992,-0.431884716383229,0.430159227344712],[0,0,0,0],[8.999999E+09,8.999999E+09,8.999999E+09,8.999999E+09,8.999999E+09,8.999999E+09]];
    LOCAL CONST Robtarget Tr_meulage_motif_1_247 := [[88.6930234375,-31.96316015625,39.5983125],[0.559429550316464,-0.561673578795992,-0.431884716383229,0.430159227344712],[0,0,0,0],[8.999999E+09,8.999999E+09,8.999999E+09,8.999999E+09,8.999999E+09,8.999999E+09]];
    LOCAL CONST Robtarget Tr_meulage_motif_1_248 := [[88.535984375,-32.55483203125,39.175421875],[0.559429550316464,-0.561673578795992,-0.431884716383229,0.430159227344712],[0,0,0,0],[8.999999E+09,8.999999E+09,8.999999E+09,8.999999E+09,8.999999E+09,8.999999E+09]];
    LOCAL CONST Robtarget Tr_meulage_motif_1_249 := [[88.246625,-33.64748046875,38.64496875],[0.559429550316464,-0.561673578795992,-0.431884716383229,0.430159227344712],[0,0,0,0],[8.999999E+09,8.999999E+09,8.999999E+09,8.999999E+09,8.999999E+09,8.999999E+09]];
    LOCAL CONST Robtarget Tr_meulage_motif_1_250 := [[88.030625,-34.4644375,38.380859375],[0.559429550316464,-0.561673578795992,-0.431884716383229,0.430159227344712],[0,0,0,0],[8.999999E+09,8.999999E+09,8.999999E+09,8.999999E+09,8.999999E+09,8.999999E+09]];
    LOCAL CONST Robtarget Tr_meulage_motif_1_251 := [[87.7926015625,-35.36553125,38.17637109375],[0.559429550316464,-0.561673578795992,-0.431884716383229,0.430159227344712],[0,0,0,0],[8.999999E+09,8.999999E+09,8.999999E+09,8.999999E+09,8.999999E+09,8.999999E+09]];
    LOCAL CONST Robtarget Tr_meulage_motif_1_252 := [[87.5421875,-36.31461328125,38.06782421875],[0.559429550316464,-0.561673578795992,-0.431884716383229,0.430159227344712],[0,0,0,0],[8.999999E+09,8.999999E+09,8.999999E+09,8.999999E+09,8.999999E+09,8.999999E+09]];
    LOCAL CONST Robtarget Tr_meulage_motif_1_253 := [[87.288953125,-37.274328125,37.9572109375],[0.559429550316464,-0.561673578795992,-0.431884716383229,0.430159227344712],[0,0,0,0],[8.999999E+09,8.999999E+09,8.999999E+09,8.999999E+09,8.999999E+09,8.999999E+09]];
    LOCAL CONST Robtarget Tr_meulage_motif_1_254 := [[87.0341015625,-38.24130859375,37.9572109375],[0.559429550316464,-0.561673578795992,-0.431884716383229,0.430159227344712],[0,0,0,0],[8.999999E+09,8.999999E+09,8.999999E+09,8.999999E+09,8.999999E+09,8.999999E+09]];
    LOCAL CONST Robtarget Tr_meulage_motif_1_255 := [[86.77925,-39.2082890625,37.95720703125],[0.559429550316464,-0.561673578795992,-0.431884716383229,0.430159227344712],[0,0,0,0],[8.999999E+09,8.999999E+09,8.999999E+09,8.999999E+09,8.999999E+09,8.999999E+09]];
    LOCAL CONST Robtarget Tr_meulage_motif_1_256 := [[86.5243984375,-40.17526953125,37.95720703125],[0.559429550316464,-0.561673578795992,-0.431884716383229,0.430159227344712],[0,0,0,0],[8.999999E+09,8.999999E+09,8.999999E+09,8.999999E+09,8.999999E+09,8.999999E+09]];
    LOCAL CONST Robtarget Tr_meulage_motif_1_257 := [[86.2695390625,-41.14224609375,37.95720703125],[0.559429550316464,-0.561673578795992,-0.431884716383229,0.430159227344712],[0,0,0,0],[8.999999E+09,8.999999E+09,8.999999E+09,8.999999E+09,8.999999E+09,8.999999E+09]];
    LOCAL CONST Robtarget Tr_meulage_motif_1_258 := [[86.0146875,-42.1092265625,37.957203125],[0.559429550316464,-0.561673578795992,-0.431884716383229,0.430159227344712],[0,0,0,0],[8.999999E+09,8.999999E+09,8.999999E+09,8.999999E+09,8.999999E+09,8.999999E+09]];
    LOCAL CONST Robtarget Tr_meulage_motif_1_259 := [[85.7598359375,-43.07620703125,37.957203125],[0.559429550316464,-0.561673578795992,-0.431884716383229,0.430159227344712],[0,0,0,0],[8.999999E+09,8.999999E+09,8.999999E+09,8.999999E+09,8.999999E+09,8.999999E+09]];
    LOCAL CONST Robtarget Tr_meulage_motif_1_260 := [[85.504984375,-44.0431875,37.95719921875],[0.559429550316464,-0.561673578795992,-0.431884716383229,0.430159227344712],[0,0,0,0],[8.999999E+09,8.999999E+09,8.999999E+09,8.999999E+09,8.999999E+09,8.999999E+09]];
    LOCAL CONST Robtarget Tr_meulage_motif_1_261 := [[85.2501328125,-45.01016796875,37.95719921875],[0.559429550316464,-0.561673578795992,-0.431884716383229,0.430159227344712],[0,0,0,0],[8.999999E+09,8.999999E+09,8.999999E+09,8.999999E+09,8.999999E+09,8.999999E+09]];
    LOCAL CONST Robtarget Tr_meulage_motif_1_262 := [[84.9952734375,-45.97714453125,37.9571953125],[0.559429550316464,-0.561673578795992,-0.431884716383229,0.430159227344712],[0,0,0,0],[8.999999E+09,8.999999E+09,8.999999E+09,8.999999E+09,8.999999E+09,8.999999E+09]];
    LOCAL CONST Robtarget Tr_meulage_motif_1_263 := [[84.740421875,-46.944125,37.9571953125],[0.559429550316464,-0.561673578795992,-0.431884716383229,0.430159227344712],[0,0,0,0],[8.999999E+09,8.999999E+09,8.999999E+09,8.999999E+09,8.999999E+09,8.999999E+09]];
    LOCAL CONST Robtarget Tr_meulage_motif_1_264 := [[84.4855703125,-47.91110546875,37.95719140625],[0.559429550316464,-0.561673578795992,-0.431884716383229,0.430159227344712],[0,0,0,0],[8.999999E+09,8.999999E+09,8.999999E+09,8.999999E+09,8.999999E+09,8.999999E+09]];
    LOCAL CONST Robtarget Tr_meulage_motif_1_265 := [[84.23071875,-48.8780859375,37.95719140625],[0.559429550316464,-0.561673578795992,-0.431884716383229,0.430159227344712],[0,0,0,0],[8.999999E+09,8.999999E+09,8.999999E+09,8.999999E+09,8.999999E+09,8.999999E+09]];
    LOCAL CONST Robtarget Tr_meulage_motif_1_266 := [[83.975859375,-49.84506640625,37.9571875],[0.559429550316464,-0.561673578795992,-0.431884716383229,0.430159227344712],[0,0,0,0],[8.999999E+09,8.999999E+09,8.999999E+09,8.999999E+09,8.999999E+09,8.999999E+09]];
    LOCAL CONST Robtarget Tr_meulage_motif_1_267 := [[83.7210078125,-50.81204296875,37.9571875],[0.559429550316464,-0.561673578795992,-0.431884716383229,0.430159227344712],[0,0,0,0],[8.999999E+09,8.999999E+09,8.999999E+09,8.999999E+09,8.999999E+09,8.999999E+09]];
    LOCAL CONST Robtarget Tr_meulage_motif_1_268 := [[83.46615625,-51.7790234375,37.95718359375],[0.559429550316464,-0.561673578795992,-0.431884716383229,0.430159227344712],[0,0,0,0],[8.999999E+09,8.999999E+09,8.999999E+09,8.999999E+09,8.999999E+09,8.999999E+09]];
    LOCAL CONST Robtarget Tr_meulage_motif_1_269 := [[83.2113046875,-52.74600390625,37.95718359375],[0.559429550316464,-0.561673578795992,-0.431884716383229,0.430159227344712],[0,0,0,0],[8.999999E+09,8.999999E+09,8.999999E+09,8.999999E+09,8.999999E+09,8.999999E+09]];
    LOCAL CONST Robtarget Tr_meulage_motif_1_270 := [[82.9564453125,-53.712984375,37.9571796875],[0.559429550316464,-0.561673578795992,-0.431884716383229,0.430159227344712],[0,0,0,0],[8.999999E+09,8.999999E+09,8.999999E+09,8.999999E+09,8.999999E+09,8.999999E+09]];
    LOCAL CONST Robtarget Tr_meulage_motif_1_271 := [[82.70159375,-54.67996484375,37.9571796875],[0.559429550316464,-0.561673578795992,-0.431884716383229,0.430159227344712],[0,0,0,0],[8.999999E+09,8.999999E+09,8.999999E+09,8.999999E+09,8.999999E+09,8.999999E+09]];
    LOCAL CONST Robtarget Tr_meulage_motif_1_272 := [[82.4467421875,-55.64694140625,37.95717578125],[0.559429550316464,-0.561673578795992,-0.431884716383229,0.430159227344712],[0,0,0,0],[8.999999E+09,8.999999E+09,8.999999E+09,8.999999E+09,8.999999E+09,8.999999E+09]];
    LOCAL CONST Robtarget Tr_meulage_motif_1_273 := [[82.191890625,-56.613921875,37.95717578125],[0.559429550316464,-0.561673578795992,-0.431884716383229,0.430159227344712],[0,0,0,0],[8.999999E+09,8.999999E+09,8.999999E+09,8.999999E+09,8.999999E+09,8.999999E+09]];
    LOCAL CONST Robtarget Tr_meulage_motif_1_274 := [[81.93703125,-57.58090234375,37.957171875],[0.559429550316464,-0.561673578795992,-0.431884716383229,0.430159227344712],[0,0,0,0],[8.999999E+09,8.999999E+09,8.999999E+09,8.999999E+09,8.999999E+09,8.999999E+09]];
    LOCAL CONST Robtarget Tr_meulage_motif_1_275 := [[81.6821796875,-58.5478828125,37.957171875],[0.559429550316464,-0.561673578795992,-0.431884716383229,0.430159227344712],[0,0,0,0],[8.999999E+09,8.999999E+09,8.999999E+09,8.999999E+09,8.999999E+09,8.999999E+09]];
    LOCAL CONST Robtarget Tr_meulage_motif_1_276 := [[81.427328125,-59.51486328125,37.95716796875],[0.559429550316464,-0.561673578795992,-0.431884716383229,0.430159227344712],[0,0,0,0],[8.999999E+09,8.999999E+09,8.999999E+09,8.999999E+09,8.999999E+09,8.999999E+09]];
    LOCAL CONST Robtarget Tr_meulage_motif_1_277 := [[81.1724765625,-60.48183984375,37.95716796875],[0.559429550316464,-0.561673578795992,-0.431884716383229,0.430159227344712],[0,0,0,0],[8.999999E+09,8.999999E+09,8.999999E+09,8.999999E+09,8.999999E+09,8.999999E+09]];
    LOCAL CONST Robtarget Tr_meulage_motif_1_278 := [[80.9176171875,-61.4488203125,37.9571640625],[0.559429550316464,-0.561673578795992,-0.431884716383229,0.430159227344712],[0,0,0,0],[8.999999E+09,8.999999E+09,8.999999E+09,8.999999E+09,8.999999E+09,8.999999E+09]];
    LOCAL CONST Robtarget Tr_meulage_motif_1_279 := [[80.662765625,-62.41580078125,37.9571640625],[0.559429550316464,-0.561673578795992,-0.431884716383229,0.430159227344712],[0,0,0,0],[8.999999E+09,8.999999E+09,8.999999E+09,8.999999E+09,8.999999E+09,8.999999E+09]];
    LOCAL CONST Robtarget Tr_meulage_motif_1_280 := [[80.4079140625,-63.38278125,37.95716015625],[0.559429550316464,-0.561673578795992,-0.431884716383229,0.430159227344712],[0,0,0,0],[8.999999E+09,8.999999E+09,8.999999E+09,8.999999E+09,8.999999E+09,8.999999E+09]];
    LOCAL CONST Robtarget Tr_meulage_motif_1_281 := [[80.1530625,-64.34976171875,37.95716015625],[0.559429550316464,-0.561673578795992,-0.431884716383229,0.430159227344712],[0,0,0,0],[8.999999E+09,8.999999E+09,8.999999E+09,8.999999E+09,8.999999E+09,8.999999E+09]];
    LOCAL CONST Robtarget Tr_meulage_motif_1_282 := [[79.8982109375,-65.31673828125,37.95715625],[0.559429550316464,-0.561673578795992,-0.431884716383229,0.430159227344712],[0,0,0,0],[8.999999E+09,8.999999E+09,8.999999E+09,8.999999E+09,8.999999E+09,8.999999E+09]];
    LOCAL CONST Robtarget Tr_meulage_motif_1_283 := [[79.6433515625,-66.28371875,37.95715625],[0.559429550316464,-0.561673578795992,-0.431884716383229,0.430159227344712],[0,0,0,0],[8.999999E+09,8.999999E+09,8.999999E+09,8.999999E+09,8.999999E+09,8.999999E+09]];
    LOCAL CONST Robtarget Tr_meulage_motif_1_284 := [[79.3885,-67.2506953125,37.95715234375],[0.559429550316464,-0.561673578795992,-0.431884716383229,0.430159227344712],[0,0,0,0],[8.999999E+09,8.999999E+09,8.999999E+09,8.999999E+09,8.999999E+09,8.999999E+09]];
    LOCAL CONST Robtarget Tr_meulage_motif_1_285 := [[79.1336484375,-68.2176796875,37.95715234375],[0.559429550316464,-0.561673578795992,-0.431884716383229,0.430159227344712],[0,0,0,0],[8.999999E+09,8.999999E+09,8.999999E+09,8.999999E+09,8.999999E+09,8.999999E+09]];
    LOCAL CONST Robtarget Tr_meulage_motif_1_286 := [[78.878796875,-69.18465625,37.9571484375],[0.559429550316464,-0.561673578795992,-0.431884716383229,0.430159227344712],[0,0,0,0],[8.999999E+09,8.999999E+09,8.999999E+09,8.999999E+09,8.999999E+09,8.999999E+09]];
    LOCAL CONST Robtarget Tr_meulage_motif_1_287 := [[78.6239375,-70.151640625,37.9571484375],[0.559429550316464,-0.561673578795992,-0.431884716383229,0.430159227344712],[0,0,0,0],[8.999999E+09,8.999999E+09,8.999999E+09,8.999999E+09,8.999999E+09,8.999999E+09]];
    LOCAL CONST Robtarget Tr_meulage_motif_1_288 := [[78.3690859375,-71.1186171875,37.95714453125],[0.559429550316464,-0.561673578795992,-0.431884716383229,0.430159227344712],[0,0,0,0],[8.999999E+09,8.999999E+09,8.999999E+09,8.999999E+09,8.999999E+09,8.999999E+09]];
    LOCAL CONST Robtarget Tr_meulage_motif_1_289 := [[78.114234375,-72.08559375,37.95714453125],[0.559429550316464,-0.561673578795992,-0.431884716383229,0.430159227344712],[0,0,0,0],[8.999999E+09,8.999999E+09,8.999999E+09,8.999999E+09,8.999999E+09,8.999999E+09]];
    LOCAL CONST Robtarget Tr_meulage_motif_1_290 := [[77.8593828125,-73.052578125,37.957140625],[0.559429550316464,-0.561673578795992,-0.431884716383229,0.430159227344712],[0,0,0,0],[8.999999E+09,8.999999E+09,8.999999E+09,8.999999E+09,8.999999E+09,8.999999E+09]];
    LOCAL CONST Robtarget Tr_meulage_motif_1_291 := [[77.6045234375,-74.0195546875,37.957140625],[0.559429550316464,-0.561673578795992,-0.431884716383229,0.430159227344712],[0,0,0,0],[8.999999E+09,8.999999E+09,8.999999E+09,8.999999E+09,8.999999E+09,8.999999E+09]];
    LOCAL CONST Robtarget Tr_meulage_motif_1_292 := [[77.349671875,-74.9865390625,37.95713671875],[0.559429550316464,-0.561673578795992,-0.431884716383229,0.430159227344712],[0,0,0,0],[8.999999E+09,8.999999E+09,8.999999E+09,8.999999E+09,8.999999E+09,8.999999E+09]];
    LOCAL CONST Robtarget Tr_meulage_motif_1_293 := [[77.0948203125,-75.953515625,37.95713671875],[0.559429550316464,-0.561673578795992,-0.431884716383229,0.430159227344712],[0,0,0,0],[8.999999E+09,8.999999E+09,8.999999E+09,8.999999E+09,8.999999E+09,8.999999E+09]];
    LOCAL CONST Robtarget Tr_meulage_motif_1_294 := [[76.83996875,-76.9204921875,37.9571328125],[0.559429550316464,-0.561673578795992,-0.431884716383229,0.430159227344712],[0,0,0,0],[8.999999E+09,8.999999E+09,8.999999E+09,8.999999E+09,8.999999E+09,8.999999E+09]];

